LIN {X 0,Y 312.63,Z 536.352,A -85,B 0,C 180,E1 -15641.656,E2 -15641.656} C_VEL
LIN {X 0,Y 312.686,Z 536.349,A -85,B 0,C 180,E1 -15645.686,E2 -15645.686} C_VEL
LIN {X 0,Y 312.696,Z 536.347,A -85,B 0,C 180,E1 -15649.642,E2 -15649.642} C_VEL
LIN {X 0,Y 312.865,Z 536.328,A -85,B 0,C 180,E1 -15652.255,E2 -15652.255} C_VEL
LIN {X 0,Y 312.73,Z 536.383,A -85,B 0,C 180,E1 -15655.005,E2 -15655.005} C_VEL
LIN {X 0,Y 312.813,Z 536.954,A -85,B 0,C 180,E1 -15655.329,E2 -15655.329} C_VEL
LIN {X 0,Y 313.996,Z 539.629,A -85,B 0,C 180,E1 -15655.654,E2 -15655.654} C_VEL
LIN {X 0,Y 315.234,Z 541.537,A -85,B 0,C 180,E1 -15655.877,E2 -15655.877} C_VEL
LIN {X 0,Y 320.48,Z 550.525,A -85,B 0,C 180,E1 -15656.823,E2 -15656.823} C_VEL
LIN {X 0,Y 324.46,Z 558.584,A -85,B 0,C 180,E1 -15657.53,E2 -15657.53} C_VEL
LIN {X 0,Y 325.877,Z 561.864,A -85,B 0,C 180,E1 -15657.785,E2 -15657.785} C_VEL
LIN {X 0,Y 325.89,Z 581.398,A -85,B 0,C 180,E1 -15658.425,E2 -15658.425} C_VEL
LIN {X 0,Y 325.629,Z 593.005,A -85,B 0,C 180,E1 -15659.034,E2 -15659.034} C_VEL
LIN {X 0,Y 325.007,Z 604.189,A -85,B 0,C 180,E1 -15659.846,E2 -15659.846} C_VEL
LIN {X 0,Y 323.968,Z 615.161,A -85,B 0,C 180,E1 -15660.872,E2 -15660.872} C_VEL
LIN {X 0,Y 322.791,Z 625.783,A -85,B 0,C 180,E1 -15662.153,E2 -15662.153} C_VEL
LIN {X 0,Y 321.588,Z 634.422,A -85,B 0,C 180,E1 -15663.446,E2 -15663.446} C_VEL
LIN {X 0,Y 320.193,Z 643.041,A -85,B 0,C 180,E1 -15665.037,E2 -15665.037} C_VEL
LIN {X 0,Y 318.928,Z 650.052,A -85,B 0,C 180,E1 -15666.64,E2 -15666.64} C_VEL
LIN {X 0,Y 317.7,Z 655.851,A -85,B 0,C 180,E1 -15668.268,E2 -15668.268} C_VEL
LIN {X 0,Y 316.44,Z 661.361,A -85,B 0,C 180,E1 -15670.235,E2 -15670.235} C_VEL
LIN {X 0,Y 315.396,Z 665.429,A -85,B 0,C 180,E1 -15672.157,E2 -15672.157} C_VEL
LIN {X 0,Y 314.468,Z 668.571,A -85,B 0,C 180,E1 -15674.232,E2 -15674.232} C_VEL
LIN {X 0,Y 313.936,Z 670.088,A -85,B 0,C 180,E1 -15675.719,E2 -15675.719} C_VEL
LIN {X 0,Y 313.56,Z 670.868,A -85,B 0,C 180,E1 -15676.941,E2 -15676.941} C_VEL
LIN {X 0,Y 313.238,Z 671.303,A -85,B 0,C 180,E1 -15678.308,E2 -15678.308} C_VEL
LIN {X 0,Y 313.012,Z 671.234,A -85,B 0,C 180,E1 -15679.682,E2 -15679.682} C_VEL
LIN {X 0,Y 312.851,Z 670.681,A -85,B 0,C 180,E1 -15681.066,E2 -15681.066} C_VEL
LIN {X 0,Y 312.748,Z 669.215,A -85,B 0,C 180,E1 -15682.881,E2 -15682.881} C_VEL
LIN {X 0,Y 312.895,Z 665.987,A -85,B 0,C 180,E1 -15685.263,E2 -15685.263} C_VEL
LIN {X 0,Y 313.204,Z 661.722,A -85,B 0,C 180,E1 -15687.388,E2 -15687.388} C_VEL
LIN {X 0,Y 313.668,Z 655.995,A -85,B 0,C 180,E1 -15689.534,E2 -15689.534} C_VEL
LIN {X 0,Y 314.243,Z 649.623,A -85,B 0,C 180,E1 -15691.402,E2 -15691.402} C_VEL
LIN {X 0,Y 314.858,Z 642.22,A -85,B 0,C 180,E1 -15693.153,E2 -15693.153} C_VEL
LIN {X 0,Y 315.63,Z 633.354,A -85,B 0,C 180,E1 -15694.86,E2 -15694.86} C_VEL
LIN {X 0,Y 316.364,Z 624.447,A -85,B 0,C 180,E1 -15696.262,E2 -15696.262} C_VEL
LIN {X 0,Y 317.032,Z 614.062,A -85,B 0,C 180,E1 -15697.592,E2 -15697.592} C_VEL
LIN {X 0,Y 317.81,Z 601.895,A -85,B 0,C 180,E1 -15698.818,E2 -15698.818} C_VEL
LIN {X 0,Y 318.333,Z 589.989,A -85,B 0,C 180,E1 -15699.733,E2 -15699.733} C_VEL
LIN {X 0,Y 318.574,Z 576.988,A -85,B 0,C 180,E1 -15700.458,E2 -15700.458} C_VEL
LIN {X 0,Y 318.669,Z 563.154,A -85,B 0,C 180,E1 -15700.946,E2 -15700.946} C_VEL
LIN {X 0,Y 318.586,Z 555.236,A -85,B 0,C 180,E1 -15701.168,E2 -15701.168} C_VEL
LIN {X 0,Y 312.709,Z 537.424,A -85,B 0,C 180,E1 -15701.948,E2 -15701.948} C_VEL
LIN {X 0,Y 312.51,Z 536.496,A -85,B 0,C 180,E1 -15702.177,E2 -15702.177} C_VEL
LIN {X 0,Y 312.536,Z 536.364,A -85,B 0,C 180,E1 -15706.021,E2 -15706.021} C_VEL
LIN {X 0,Y 312.53,Z 536.366,A -85,B 0,C 180,E1 -15709.87,E2 -15709.87} C_VEL
LIN {X 0,Y 312.552,Z 536.362,A -85,B 0,C 180,E1 -15712.62,E2 -15712.62} C_VEL
LIN {X 0,Y 312.52,Z 536.366,A -85,B 0,C 180,E1 -15716.312,E2 -15716.312} C_VEL
LIN {X 0,Y 312.547,Z 536.362,A -85,B 0,C 180,E1 -15720.351,E2 -15720.351} C_VEL
LIN {X 0,Y 312.605,Z 536.356,A -85,B 0,C 180,E1 -15724.065,E2 -15724.065} C_VEL
LIN {X 0,Y 312.59,Z 536.362,A -85,B 0,C 180,E1 -15727.53,E2 -15727.53} C_VEL
LIN {X 0,Y 312.585,Z 536.362,A -85,B 0,C 180,E1 -15731.654,E2 -15731.654} C_VEL
LIN {X 0,Y 312.689,Z 536.349,A -85,B 0,C 180,E1 -15735.686,E2 -15735.686} C_VEL
LIN {X 0,Y 312.702,Z 536.349,A -85,B 0,C 180,E1 -15739.642,E2 -15739.642} C_VEL
LIN {X 0,Y 312.821,Z 536.328,A -85,B 0,C 180,E1 -15742.253,E2 -15742.253} C_VEL
LIN {X 0,Y 312.71,Z 536.342,A -85,B 0,C 180,E1 -15744.842,E2 -15744.842} C_VEL
LIN {X 0,Y 312.993,Z 536.306,A -85,B 0,C 180,E1 -15748.713,E2 -15748.713} C_VEL
LIN {X 0,Y 312.993,Z 536.308,A -85,B 0,C 180,E1 -15751.287,E2 -15751.287} C_VEL
LIN {X 0,Y 312.71,Z 536.342,A -85,B 0,C 180,E1 -15755.158,E2 -15755.158} C_VEL
LIN {X 0,Y 312.822,Z 536.333,A -85,B 0,C 180,E1 -15757.747,E2 -15757.747} C_VEL
LIN {X 0,Y 312.668,Z 536.351,A -85,B 0,C 180,E1 -15761.671,E2 -15761.671} C_VEL
LIN {X 0,Y 312.704,Z 536.342,A -85,B 0,C 180,E1 -15764.887,E2 -15764.887} C_VEL
LIN {X 0,Y 312.633,Z 536.352,A -85,B 0,C 180,E1 -15769.235,E2 -15769.235} C_VEL
LIN {X 0,Y 312.529,Z 536.364,A -85,B 0,C 180,E1 -15772.78,E2 -15772.78} C_VEL
LIN {X 0,Y 312.605,Z 536.361,A -85,B 0,C 180,E1 -15775.935,E2 -15775.935} C_VEL
LIN {X 0,Y 312.54,Z 536.365,A -85,B 0,C 180,E1 -15779.65,E2 -15779.65} C_VEL
LIN {X 0,Y 312.521,Z 536.368,A -85,B 0,C 180,E1 -15783.688,E2 -15783.688} C_VEL
LIN {X 0,Y 312.553,Z 536.361,A -85,B 0,C 180,E1 -15787.38,E2 -15787.38} C_VEL
LIN {X 0,Y 312.533,Z 536.365,A -85,B 0,C 180,E1 -15790.701,E2 -15790.701} C_VEL
LIN {X 0,Y 312.536,Z 536.368,A -85,B 0,C 180,E1 -15794.193,E2 -15794.193} C_VEL
LIN {X 0,Y 312.485,Z 536.373,A -85,B 0,C 180,E1 -15797.917,E2 -15797.917} C_VEL
LIN {X 0,Y 312.532,Z 536.367,A -85,B 0,C 180,E1 -15801.909,E2 -15801.909} C_VEL
LIN {X 0,Y 312.504,Z 536.369,A -85,B 0,C 180,E1 -15805.789,E2 -15805.789} C_VEL
LIN {X 0,Y 312.525,Z 536.365,A -85,B 0,C 180,E1 -15808.853,E2 -15808.853} C_VEL
LIN {X 0,Y 312.543,Z 536.361,A -85,B 0,C 180,E1 -15812.28,E2 -15812.28} C_VEL
LIN {X 0,Y 312.581,Z 536.359,A -85,B 0,C 180,E1 -15814.71,E2 -15814.71} C_VEL
LIN {X 0,Y 312.559,Z 536.359,A -85,B 0,C 180,E1 -15817.877,E2 -15817.877} C_VEL
LIN {X 0,Y 311.858,Z 536.449,A -85,B 0,C 180,E1 -15818.953,E2 -15818.953} C_VEL
LIN {X 0,Y 309.002,Z 536.806,A -85,B 0,C 180,E1 -15820.705,E2 -15820.705} C_VEL
LIN {X 0,Y 306.622,Z 537.103,A -85,B 0,C 180,E1 -15822.125,E2 -15822.125} C_VEL
LIN {X 0,Y 305.631,Z 537.223,A -85,B 0,C 180,E1 -15823.225,E2 -15823.225} C_VEL
LIN {X 0,Y 305.566,Z 537.232,A -85,B 0,C 180,E1 -15823.597,E2 -15823.597} C_VEL
LIN {X 0,Y 305.585,Z 537.232,A -85,B 0,C 180,E1 -15826.703,E2 -15826.703} C_VEL
LIN {X 0,Y 305.791,Z 537.203,A -85,B 0,C 180,E1 -15831.207,E2 -15831.207} C_VEL
LIN {X 0,Y 305.847,Z 537.196,A -85,B 0,C 180,E1 -15833.402,E2 -15833.402} C_VEL
LIN {X 0,Y 305.951,Z 537.187,A -85,B 0,C 180,E1 -15838.683,E2 -15838.683} C_VEL
LIN {X 0,Y 305.95,Z 537.184,A -85,B 0,C 180,E1 -15841.316,E2 -15841.316} C_VEL
LIN {X 0,Y 305.682,Z 537.218,A -85,B 0,C 180,E1 -15845.276,E2 -15845.276} C_VEL
LIN {X 0,Y 305.802,Z 537.203,A -85,B 0,C 180,E1 -15847.926,E2 -15847.926} C_VEL
LIN {X 0,Y 305.596,Z 537.228,A -85,B 0,C 180,E1 -15851.945,E2 -15851.945} C_VEL
LIN {X 0,Y 305.631,Z 537.225,A -85,B 0,C 180,E1 -15855.034,E2 -15855.034} C_VEL
LIN {X 0,Y 305.573,Z 537.235,A -85,B 0,C 180,E1 -15858.783,E2 -15858.783} C_VEL
LIN {X 0,Y 305.48,Z 537.245,A -85,B 0,C 180,E1 -15863.039,E2 -15863.039} C_VEL
LIN {X 0,Y 305.548,Z 537.235,A -85,B 0,C 180,E1 -15866.229,E2 -15866.229} C_VEL
LIN {X 0,Y 305.49,Z 537.244,A -85,B 0,C 180,E1 -15869.05,E2 -15869.05} C_VEL
LIN {X 0,Y 305.459,Z 537.245,A -85,B 0,C 180,E1 -15873.517,E2 -15873.517} C_VEL
LIN {X 0,Y 305.467,Z 537.249,A -85,B 0,C 180,E1 -15876.74,E2 -15876.74} C_VEL
LIN {X 0,Y 305.449,Z 537.25,A -85,B 0,C 180,E1 -15880.6,E2 -15880.6} C_VEL
LIN {X 0,Y 305.414,Z 537.253,A -85,B 0,C 180,E1 -15884.493,E2 -15884.493} C_VEL
LIN {X 0,Y 305.438,Z 537.248,A -85,B 0,C 180,E1 -15888.144,E2 -15888.144} C_VEL
LIN {X 0,Y 305.472,Z 537.244,A -85,B 0,C 180,E1 -15891.598,E2 -15891.598} C_VEL
LIN {X 0,Y 305.61,Z 537.416,A -85,B 0,C 180,E1 -15894.301,E2 -15894.301} C_VEL
LIN {X 0,Y 308.315,Z 551.362,A -85,B 0,C 180,E1 -15898.752,E2 -15898.752} C_VEL
LIN {X 0,Y 309.128,Z 556.658,A -85,B 0,C 180,E1 -15900.365,E2 -15900.365} C_VEL
LIN {X 0,Y 307.296,Z 571.295,A -85,B 0,C 180,E1 -15904.608,E2 -15904.608} C_VEL
LIN {X 0,Y 305.685,Z 588.18,A -85,B 0,C 180,E1 -15909.476,E2 -15909.476} C_VEL
LIN {X 0,Y 305.517,Z 589.903,A -85,B 0,C 180,E1 -15909.891,E2 -15909.891} C_VEL
LIN {X 0,Y 309.829,Z 651.427,A -85,B 0,C 180,E1 -15912.133,E2 -15912.133} C_VEL
LIN {X 0,Y 309.126,Z 676.197,A -85,B 0,C 180,E1 -15912.98,E2 -15912.98} C_VEL
LIN {X 0,Y 308.596,Z 687.867,A -85,B 0,C 180,E1 -15913.631,E2 -15913.631} C_VEL
LIN {X 0,Y 307.713,Z 698.277,A -85,B 0,C 180,E1 -15914.433,E2 -15914.433} C_VEL
LIN {X 0,Y 306.771,Z 709.39,A -85,B 0,C 180,E1 -15915.574,E2 -15915.574} C_VEL
LIN {X 0,Y 306.007,Z 719.359,A -85,B 0,C 180,E1 -15916.892,E2 -15916.892} C_VEL
LIN {X 0,Y 305.232,Z 728.218,A -85,B 0,C 180,E1 -15918.377,E2 -15918.377} C_VEL
LIN {X 0,Y 304.777,Z 736.134,A -85,B 0,C 180,E1 -15920.041,E2 -15920.041} C_VEL
LIN {X 0,Y 304.572,Z 742.449,A -85,B 0,C 180,E1 -15921.708,E2 -15921.708} C_VEL
LIN {X 0,Y 304.624,Z 747.486,A -85,B 0,C 180,E1 -15923.376,E2 -15923.376} C_VEL
LIN {X 0,Y 304.895,Z 752.023,A -85,B 0,C 180,E1 -15925.373,E2 -15925.373} C_VEL
LIN {X 0,Y 305.09,Z 755.096,A -85,B 0,C 180,E1 -15927.359,E2 -15927.359} C_VEL
LIN {X 0,Y 305.334,Z 756.407,A -85,B 0,C 180,E1 -15928.681,E2 -15928.681} C_VEL
LIN {X 0,Y 305.562,Z 757.164,A -85,B 0,C 180,E1 -15930,E2 -15930} C_VEL
LIN {X 0,Y 305.109,Z 757.234,A -85,B 0,C 180,E1 -15931.32,E2 -15931.32} C_VEL
LIN {X 0,Y 304.892,Z 756.821,A -85,B 0,C 180,E1 -15932.642,E2 -15932.642} C_VEL
LIN {X 0,Y 304.681,Z 755.839,A -85,B 0,C 180,E1 -15933.968,E2 -15933.968} C_VEL
LIN {X 0,Y 304.419,Z 754.339,A -85,B 0,C 180,E1 -15935.298,E2 -15935.298} C_VEL
LIN {X 0,Y 304.248,Z 751.04,A -85,B 0,C 180,E1 -15937.299,E2 -15937.299} C_VEL
LIN {X 0,Y 304.4,Z 746.467,A -85,B 0,C 180,E1 -15939.3,E2 -15939.3} C_VEL
LIN {X 0,Y 304.897,Z 740.46,A -85,B 0,C 180,E1 -15941.299,E2 -15941.299} C_VEL
LIN {X 0,Y 305.993,Z 732.774,A -85,B 0,C 180,E1 -15943.278,E2 -15943.278} C_VEL
LIN {X 0,Y 307.358,Z 724.75,A -85,B 0,C 180,E1 -15944.906,E2 -15944.906} C_VEL
LIN {X 0,Y 308.946,Z 714.928,A -85,B 0,C 180,E1 -15946.52,E2 -15946.52} C_VEL
LIN {X 0,Y 310.94,Z 703.756,A -85,B 0,C 180,E1 -15947.936,E2 -15947.936} C_VEL
LIN {X 0,Y 312.695,Z 691.885,A -85,B 0,C 180,E1 -15949.096,E2 -15949.096} C_VEL
LIN {X 0,Y 314.143,Z 680.329,A -85,B 0,C 180,E1 -15949.948,E2 -15949.948} C_VEL
LIN {X 0,Y 315.4,Z 667.35,A -85,B 0,C 180,E1 -15950.63,E2 -15950.63} C_VEL
LIN {X 0,Y 316.09,Z 651.138,A -85,B 0,C 180,E1 -15951.19,E2 -15951.19} C_VEL
LIN {X 0,Y 315.177,Z 625.529,A -85,B 0,C 180,E1 -15952.203,E2 -15952.203} C_VEL
LIN {X 0,Y 313.343,Z 607.824,A -85,B 0,C 180,E1 -15953.06,E2 -15953.06} C_VEL
LIN {X 0,Y 310.491,Z 589.45,A -85,B 0,C 180,E1 -15954.097,E2 -15954.097} C_VEL
LIN {X 0,Y 307.119,Z 572.651,A -85,B 0,C 180,E1 -15955.24,E2 -15955.24} C_VEL
LIN {X 0,Y 307.26,Z 570.491,A -85,B 0,C 180,E1 -15955.758,E2 -15955.758} C_VEL
LIN {X 0,Y 309.042,Z 557.571,A -85,B 0,C 180,E1 -15959.644,E2 -15959.644} C_VEL
LIN {X 0,Y 309.131,Z 555.676,A -85,B 0,C 180,E1 -15960.241,E2 -15960.241} C_VEL
LIN {X 0,Y 307.588,Z 547.039,A -85,B 0,C 180,E1 -15963.254,E2 -15963.254} C_VEL
LIN {X 0,Y 305.816,Z 538.651,A -85,B 0,C 180,E1 -15966.454,E2 -15966.454} C_VEL
LIN {X 0,Y 305.495,Z 537.259,A -85,B 0,C 180,E1 -15967.148,E2 -15967.148} C_VEL
LIN {X 0,Y 305.45,Z 537.248,A -85,B 0,C 180,E1 -15970.599,E2 -15970.599} C_VEL
LIN {X 0,Y 305.456,Z 537.244,A -85,B 0,C 180,E1 -15974.5,E2 -15974.5} C_VEL
LIN {X 0,Y 305.49,Z 537.236,A -85,B 0,C 180,E1 -15978.152,E2 -15978.152} C_VEL
LIN {X 0,Y 305.516,Z 537.236,A -85,B 0,C 180,E1 -15981.604,E2 -15981.604} C_VEL
LIN {X 0,Y 305.457,Z 537.243,A -85,B 0,C 180,E1 -15984.887,E2 -15984.887} C_VEL
LIN {X 0,Y 305.45,Z 537.246,A -85,B 0,C 180,E1 -15988.353,E2 -15988.353} C_VEL
LIN {X 0,Y 305.514,Z 537.236,A -85,B 0,C 180,E1 -15991.114,E2 -15991.114} C_VEL
LIN {X 0,Y 305.564,Z 537.228,A -85,B 0,C 180,E1 -15994.088,E2 -15994.088} C_VEL
LIN {X 0,Y 305.518,Z 537.243,A -85,B 0,C 180,E1 -15998.405,E2 -15998.405} C_VEL
LIN {X 0,Y 305.582,Z 537.233,A -85,B 0,C 180,E1 -16001.218,E2 -16001.218} C_VEL
LIN {X 0,Y 305.642,Z 537.224,A -85,B 0,C 180,E1 -16005.349,E2 -16005.349} C_VEL
LIN {X 0,Y 305.633,Z 537.226,A -85,B 0,C 180,E1 -16009.4,E2 -16009.4} C_VEL
LIN {X 0,Y 305.806,Z 537.209,A -85,B 0,C 180,E1 -16012.075,E2 -16012.075} C_VEL
LIN {X 0,Y 305.788,Z 537.423,A -85,B 0,C 180,E1 -16014.23,E2 -16014.23} C_VEL
LIN {X 0,Y 306.003,Z 538.467,A -85,B 0,C 180,E1 -16014.482,E2 -16014.482} C_VEL
LIN {X 0,Y 307.548,Z 541.21,A -85,B 0,C 180,E1 -16014.816,E2 -16014.816} C_VEL
LIN {X 0,Y 315.14,Z 554.13,A -85,B 0,C 180,E1 -16016.28,E2 -16016.28} C_VEL
LIN {X 0,Y 319.195,Z 562.569,A -85,B 0,C 180,E1 -16017.048,E2 -16017.048} C_VEL
LIN {X 0,Y 319.98,Z 564.66,A -85,B 0,C 180,E1 -16017.207,E2 -16017.207} C_VEL
LIN {X 0,Y 319.783,Z 583.237,A -85,B 0,C 180,E1 -16017.83,E2 -16017.83} C_VEL
LIN {X 0,Y 319.495,Z 595.045,A -85,B 0,C 180,E1 -16018.48,E2 -16018.48} C_VEL
LIN {X 0,Y 318.734,Z 606.808,A -85,B 0,C 180,E1 -16019.369,E2 -16019.369} C_VEL
LIN {X 0,Y 317.66,Z 617.762,A -85,B 0,C 180,E1 -16020.445,E2 -16020.445} C_VEL
LIN {X 0,Y 316.271,Z 628.744,A -85,B 0,C 180,E1 -16021.847,E2 -16021.847} C_VEL
LIN {X 0,Y 314.988,Z 637.224,A -85,B 0,C 180,E1 -16023.198,E2 -16023.198} C_VEL
LIN {X 0,Y 313.504,Z 645.53,A -85,B 0,C 180,E1 -16024.823,E2 -16024.823} C_VEL
LIN {X 0,Y 311.884,Z 653.43,A -85,B 0,C 180,E1 -16026.772,E2 -16026.772} C_VEL
LIN {X 0,Y 310.642,Z 658.865,A -85,B 0,C 180,E1 -16028.457,E2 -16028.457} C_VEL
LIN {X 0,Y 309.372,Z 663.964,A -85,B 0,C 180,E1 -16030.471,E2 -16030.471} C_VEL
LIN {X 0,Y 308.274,Z 667.778,A -85,B 0,C 180,E1 -16032.509,E2 -16032.509} C_VEL
LIN {X 0,Y 307.341,Z 670.417,A -85,B 0,C 180,E1 -16034.569,E2 -16034.569} C_VEL
LIN {X 0,Y 306.863,Z 671.556,A -85,B 0,C 180,E1 -16035.953,E2 -16035.953} C_VEL
LIN {X 0,Y 306.466,Z 672.239,A -85,B 0,C 180,E1 -16037.345,E2 -16037.345} C_VEL
LIN {X 0,Y 305.989,Z 672.269,A -85,B 0,C 180,E1 -16039.666,E2 -16039.666} C_VEL
LIN {X 0,Y 305.78,Z 671.318,A -85,B 0,C 180,E1 -16041.577,E2 -16041.577} C_VEL
LIN {X 0,Y 305.721,Z 669.883,A -85,B 0,C 180,E1 -16043.146,E2 -16043.146} C_VEL
LIN {X 0,Y 305.846,Z 667.094,A -85,B 0,C 180,E1 -16045.158,E2 -16045.158} C_VEL
LIN {X 0,Y 306.167,Z 662.831,A -85,B 0,C 180,E1 -16047.329,E2 -16047.329} C_VEL
LIN {X 0,Y 306.592,Z 657.404,A -85,B 0,C 180,E1 -16049.419,E2 -16049.419} C_VEL
LIN {X 0,Y 307.165,Z 650.979,A -85,B 0,C 180,E1 -16051.368,E2 -16051.368} C_VEL
LIN {X 0,Y 307.817,Z 643.311,A -85,B 0,C 180,E1 -16053.228,E2 -16053.228} C_VEL
LIN {X 0,Y 308.674,Z 633.551,A -85,B 0,C 180,E1 -16055.133,E2 -16055.133} C_VEL
LIN {X 0,Y 309.592,Z 622.854,A -85,B 0,C 180,E1 -16056.78,E2 -16056.78} C_VEL
LIN {X 0,Y 310.269,Z 612.085,A -85,B 0,C 180,E1 -16058.116,E2 -16058.116} C_VEL
LIN {X 0,Y 310.974,Z 600.262,A -85,B 0,C 180,E1 -16059.258,E2 -16059.258} C_VEL
LIN {X 0,Y 311.422,Z 588.721,A -85,B 0,C 180,E1 -16060.114,E2 -16060.114} C_VEL
LIN {X 0,Y 311.681,Z 575.777,A -85,B 0,C 180,E1 -16060.806,E2 -16060.806} C_VEL
LIN {X 0,Y 311.662,Z 556.495,A -85,B 0,C 180,E1 -16061.429,E2 -16061.429} C_VEL
LIN {X 0,Y 305.662,Z 538.299,A -85,B 0,C 180,E1 -16062.251,E2 -16062.251} C_VEL
LIN {X 0,Y 305.469,Z 537.331,A -85,B 0,C 180,E1 -16062.517,E2 -16062.517} C_VEL
LIN {X 0,Y 305.492,Z 537.242,A -85,B 0,C 180,E1 -16066.358,E2 -16066.358} C_VEL
LIN {X 0,Y 305.484,Z 537.244,A -85,B 0,C 180,E1 -16069.898,E2 -16069.898} C_VEL
LIN {X 0,Y 305.502,Z 537.244,A -85,B 0,C 180,E1 -16073.627,E2 -16073.627} C_VEL
LIN {X 0,Y 305.465,Z 537.244,A -85,B 0,C 180,E1 -16076.484,E2 -16076.484} C_VEL
LIN {X 0,Y 305.497,Z 537.241,A -85,B 0,C 180,E1 -16080.951,E2 -16080.951} C_VEL
LIN {X 0,Y 305.574,Z 537.232,A -85,B 0,C 180,E1 -16084.089,E2 -16084.089} C_VEL
LIN {X 0,Y 305.497,Z 537.24,A -85,B 0,C 180,E1 -16088.403,E2 -16088.403} C_VEL
LIN {X 0,Y 305.546,Z 537.236,A -85,B 0,C 180,E1 -16091.215,E2 -16091.215} C_VEL
LIN {X 0,Y 305.63,Z 537.226,A -85,B 0,C 180,E1 -16095.349,E2 -16095.349} C_VEL
LIN {X 0,Y 305.639,Z 537.226,A -85,B 0,C 180,E1 -16099.4,E2 -16099.4} C_VEL
LIN {X 0,Y 305.768,Z 537.208,A -85,B 0,C 180,E1 -16102.073,E2 -16102.073} C_VEL
LIN {X 0,Y 305.678,Z 537.217,A -85,B 0,C 180,E1 -16104.724,E2 -16104.724} C_VEL
LIN {X 0,Y 305.96,Z 537.182,A -85,B 0,C 180,E1 -16108.684,E2 -16108.684} C_VEL
LIN {X 0,Y 305.96,Z 537.184,A -85,B 0,C 180,E1 -16111.316,E2 -16111.316} C_VEL
LIN {X 0,Y 305.679,Z 537.219,A -85,B 0,C 180,E1 -16115.277,E2 -16115.277} C_VEL
LIN {X 0,Y 305.768,Z 537.211,A -85,B 0,C 180,E1 -16117.927,E2 -16117.927} C_VEL
LIN {X 0,Y 305.603,Z 537.232,A -85,B 0,C 180,E1 -16121.945,E2 -16121.945} C_VEL
LIN {X 0,Y 305.642,Z 537.222,A -85,B 0,C 180,E1 -16125.035,E2 -16125.035} C_VEL
LIN {X 0,Y 305.579,Z 537.231,A -85,B 0,C 180,E1 -16129.444,E2 -16129.444} C_VEL
LIN {X 0,Y 305.489,Z 537.241,A -85,B 0,C 180,E1 -16133.039,E2 -16133.039} C_VEL
LIN {X 0,Y 305.534,Z 537.238,A -85,B 0,C 180,E1 -16136.22,E2 -16136.22} C_VEL
LIN {X 0,Y 305.49,Z 537.241,A -85,B 0,C 180,E1 -16139.046,E2 -16139.046} C_VEL
LIN {X 0,Y 305.445,Z 537.252,A -85,B 0,C 180,E1 -16141.951,E2 -16141.951} C_VEL
LIN {X 0,Y 305.463,Z 537.244,A -85,B 0,C 180,E1 -16145.112,E2 -16145.112} C_VEL
LIN {X 0,Y 305.494,Z 537.242,A -85,B 0,C 180,E1 -16148.538,E2 -16148.538} C_VEL
LIN {X 0,Y 305.51,Z 537.24,A -85,B 0,C 180,E1 -16152.596,E2 -16152.596} C_VEL
LIN {X 0,Y 305.466,Z 537.247,A -85,B 0,C 180,E1 -16156.351,E2 -16156.351} C_VEL
LIN {X 0,Y 305.456,Z 537.248,A -85,B 0,C 180,E1 -16159.891,E2 -16159.891} C_VEL
LIN {X 0,Y 305.481,Z 537.243,A -85,B 0,C 180,E1 -16163.63,E2 -16163.63} C_VEL
LIN {X 0,Y 305.463,Z 537.247,A -85,B 0,C 180,E1 -16166.482,E2 -16166.482} C_VEL
LIN {X 0,Y 305.463,Z 537.245,A -85,B 0,C 180,E1 -16169.59,E2 -16169.59} C_VEL
LIN {X 0,Y 305.518,Z 537.24,A -85,B 0,C 180,E1 -16172.608,E2 -16172.608} C_VEL
LIN {X 0,Y 305.504,Z 537.239,A -85,B 0,C 180,E1 -16175.538,E2 -16175.538} C_VEL
LIN {X 0,Y 305.525,Z 537.238,A -85,B 0,C 180,E1 -16179.815,E2 -16179.815} C_VEL
LIN {X 0,Y 305.57,Z 537.234,A -85,B 0,C 180,E1 -16182.602,E2 -16182.602} C_VEL
LIN {X 0,Y 305.566,Z 537.232,A -85,B 0,C 180,E1 -16183.597,E2 -16183.597} C_VEL
LIN {X 0,Y 304.937,Z 537.314,A -85,B 0,C 180,E1 -16184.697,E2 -16184.697} C_VEL
LIN {X 0,Y 302.1,Z 537.668,A -85,B 0,C 180,E1 -16186.488,E2 -16186.488} C_VEL
LIN {X 0,Y 299.685,Z 537.967,A -85,B 0,C 180,E1 -16187.94,E2 -16187.94} C_VEL
LIN {X 0,Y 298.666,Z 538.092,A -85,B 0,C 180,E1 -16189.066,E2 -16189.066} C_VEL
LIN {X 0,Y 298.594,Z 538.099,A -85,B 0,C 180,E1 -16189.447,E2 -16189.447} C_VEL
LIN {X 0,Y 298.753,Z 538.081,A -85,B 0,C 180,E1 -16191.885,E2 -16191.885} C_VEL
LIN {X 0,Y 298.655,Z 538.097,A -85,B 0,C 180,E1 -16194.598,E2 -16194.598} C_VEL
LIN {X 0,Y 298.917,Z 538.063,A -85,B 0,C 180,E1 -16198.652,E2 -16198.652} C_VEL
LIN {X 0,Y 298.917,Z 538.06,A -85,B 0,C 180,E1 -16201.347,E2 -16201.347} C_VEL
LIN {X 0,Y 298.786,Z 538.079,A -85,B 0,C 180,E1 -16206.754,E2 -16206.754} C_VEL
LIN {X 0,Y 298.674,Z 538.089,A -85,B 0,C 180,E1 -16209.48,E2 -16209.48} C_VEL
LIN {X 0,Y 298.545,Z 538.106,A -85,B 0,C 180,E1 -16213.615,E2 -16213.615} C_VEL
LIN {X 0,Y 298.542,Z 538.11,A -85,B 0,C 180,E1 -16216.409,E2 -16216.409} C_VEL
LIN {X 0,Y 298.492,Z 538.112,A -85,B 0,C 180,E1 -16219.647,E2 -16219.647} C_VEL
LIN {X 0,Y 298.423,Z 538.122,A -85,B 0,C 180,E1 -16223.6,E2 -16223.6} C_VEL
LIN {X 0,Y 298.486,Z 538.117,A -85,B 0,C 180,E1 -16226.574,E2 -16226.574} C_VEL
LIN {X 0,Y 298.415,Z 538.122,A -85,B 0,C 180,E1 -16229.641,E2 -16229.641} C_VEL
LIN {X 0,Y 298.39,Z 538.131,A -85,B 0,C 180,E1 -16232.8,E2 -16232.8} C_VEL
LIN {X 0,Y 298.439,Z 538.124,A -85,B 0,C 180,E1 -16236.807,E2 -16236.807} C_VEL
LIN {X 0,Y 298.383,Z 538.13,A -85,B 0,C 180,E1 -16241.088,E2 -16241.088} C_VEL
LIN {X 0,Y 298.384,Z 538.13,A -85,B 0,C 180,E1 -16245.042,E2 -16245.042} C_VEL
LIN {X 0,Y 298.384,Z 538.132,A -85,B 0,C 180,E1 -16248.912,E2 -16248.912} C_VEL
LIN {X 0,Y 298.475,Z 538.12,A -85,B 0,C 180,E1 -16253.185,E2 -16253.185} C_VEL
LIN {X 0,Y 298.562,Z 538.263,A -85,B 0,C 180,E1 -16254.129,E2 -16254.129} C_VEL
LIN {X 0,Y 301.267,Z 552.322,A -85,B 0,C 180,E1 -16258.732,E2 -16258.732} C_VEL
LIN {X 0,Y 302.049,Z 556.84,A -85,B 0,C 180,E1 -16260.148,E2 -16260.148} C_VEL
LIN {X 0,Y 300.448,Z 569.706,A -85,B 0,C 180,E1 -16263.986,E2 -16263.986} C_VEL
LIN {X 0,Y 298.8,Z 585.325,A -85,B 0,C 180,E1 -16268.619,E2 -16268.619} C_VEL
LIN {X 0,Y 298.551,Z 588.735,A -85,B 0,C 180,E1 -16269.546,E2 -16269.546} C_VEL
LIN {X 0,Y 302.841,Z 651.586,A -85,B 0,C 180,E1 -16271.899,E2 -16271.899} C_VEL
LIN {X 0,Y 302.123,Z 675.368,A -85,B 0,C 180,E1 -16272.747,E2 -16272.747} C_VEL
LIN {X 0,Y 301.618,Z 686.939,A -85,B 0,C 180,E1 -16273.415,E2 -16273.415} C_VEL
LIN {X 0,Y 300.747,Z 697.315,A -85,B 0,C 180,E1 -16274.237,E2 -16274.237} C_VEL
LIN {X 0,Y 299.754,Z 708.387,A -85,B 0,C 180,E1 -16275.402,E2 -16275.402} C_VEL
LIN {X 0,Y 299.076,Z 717.224,A -85,B 0,C 180,E1 -16276.582,E2 -16276.582} C_VEL
LIN {X 0,Y 298.264,Z 726.3,A -85,B 0,C 180,E1 -16278.102,E2 -16278.102} C_VEL
LIN {X 0,Y 297.75,Z 734.414,A -85,B 0,C 180,E1 -16279.803,E2 -16279.803} C_VEL
LIN {X 0,Y 297.534,Z 742,A -85,B 0,C 180,E1 -16281.852,E2 -16281.852} C_VEL
LIN {X 0,Y 297.663,Z 747.732,A -85,B 0,C 180,E1 -16283.901,E2 -16283.901} C_VEL
LIN {X 0,Y 297.927,Z 751.908,A -85,B 0,C 180,E1 -16285.942,E2 -16285.942} C_VEL
LIN {X 0,Y 298.059,Z 753.847,A -85,B 0,C 180,E1 -16287.297,E2 -16287.297} C_VEL
LIN {X 0,Y 298.314,Z 755.241,A -85,B 0,C 180,E1 -16288.65,E2 -16288.65} C_VEL
LIN {X 0,Y 298.54,Z 756.035,A -85,B 0,C 180,E1 -16290,E2 -16290} C_VEL
LIN {X 0,Y 298.072,Z 756.178,A -85,B 0,C 180,E1 -16291.351,E2 -16291.351} C_VEL
LIN {X 0,Y 297.835,Z 755.797,A -85,B 0,C 180,E1 -16292.705,E2 -16292.705} C_VEL
LIN {X 0,Y 297.602,Z 754.888,A -85,B 0,C 180,E1 -16294.062,E2 -16294.062} C_VEL
LIN {X 0,Y 297.33,Z 753.432,A -85,B 0,C 180,E1 -16295.425,E2 -16295.425} C_VEL
LIN {X 0,Y 297.165,Z 750.26,A -85,B 0,C 180,E1 -16297.474,E2 -16297.474} C_VEL
LIN {X 0,Y 297.33,Z 745.776,A -85,B 0,C 180,E1 -16299.524,E2 -16299.524} C_VEL
LIN {X 0,Y 297.885,Z 739.902,A -85,B 0,C 180,E1 -16301.568,E2 -16301.568} C_VEL
LIN {X 0,Y 299.063,Z 732.406,A -85,B 0,C 180,E1 -16303.591,E2 -16303.591} C_VEL
LIN {X 0,Y 300.502,Z 724.661,A -85,B 0,C 180,E1 -16305.254,E2 -16305.254} C_VEL
LIN {X 0,Y 302.164,Z 715.054,A -85,B 0,C 180,E1 -16306.902,E2 -16306.902} C_VEL
LIN {X 0,Y 304.23,Z 704.239,A -85,B 0,C 180,E1 -16308.345,E2 -16308.345} C_VEL
LIN {X 0,Y 305.931,Z 693.671,A -85,B 0,C 180,E1 -16309.46,E2 -16309.46} C_VEL
LIN {X 0,Y 307.691,Z 681.024,A -85,B 0,C 180,E1 -16310.473,E2 -16310.473} C_VEL
LIN {X 0,Y 309.071,Z 668.287,A -85,B 0,C 180,E1 -16311.204,E2 -16311.204} C_VEL
LIN {X 0,Y 309.914,Z 655.245,A -85,B 0,C 180,E1 -16311.708,E2 -16311.708} C_VEL
LIN {X 0,Y 309.25,Z 629.64,A -85,B 0,C 180,E1 -16312.726,E2 -16312.726} C_VEL
LIN {X 0,Y 307.774,Z 612.039,A -85,B 0,C 180,E1 -16313.565,E2 -16313.565} C_VEL
LIN {X 0,Y 304.89,Z 592.145,A -85,B 0,C 180,E1 -16314.733,E2 -16314.733} C_VEL
LIN {X 0,Y 301.258,Z 574.403,A -85,B 0,C 180,E1 -16315.977,E2 -16315.977} C_VEL
LIN {X 0,Y 300.477,Z 570.14,A -85,B 0,C 180,E1 -16316.336,E2 -16316.336} C_VEL
LIN {X 0,Y 302.158,Z 558.138,A -85,B 0,C 180,E1 -16320.004,E2 -16320.004} C_VEL
LIN {X 0,Y 301.589,Z 553.455,A -85,B 0,C 180,E1 -16321.622,E2 -16321.622} C_VEL
LIN {X 0,Y 299.704,Z 543.654,A -85,B 0,C 180,E1 -16325.304,E2 -16325.304} C_VEL
LIN {X 0,Y 298.465,Z 538.144,A -85,B 0,C 180,E1 -16327.654,E2 -16327.654} C_VEL
LIN {X 0,Y 298.382,Z 538.131,A -85,B 0,C 180,E1 -16331.261,E2 -16331.261} C_VEL
LIN {X 0,Y 298.412,Z 538.12,A -85,B 0,C 180,E1 -16335.046,E2 -16335.046} C_VEL
LIN {X 0,Y 298.449,Z 538.117,A -85,B 0,C 180,E1 -16338.75,E2 -16338.75} C_VEL
LIN {X 0,Y 298.444,Z 538.121,A -85,B 0,C 180,E1 -16342.247,E2 -16342.247} C_VEL
LIN {X 0,Y 298.403,Z 538.128,A -85,B 0,C 180,E1 -16345.581,E2 -16345.581} C_VEL
LIN {X 0,Y 298.393,Z 538.128,A -85,B 0,C 180,E1 -16348.791,E2 -16348.791} C_VEL
LIN {X 0,Y 298.457,Z 538.121,A -85,B 0,C 180,E1 -16351.904,E2 -16351.904} C_VEL
LIN {X 0,Y 298.479,Z 538.117,A -85,B 0,C 180,E1 -16354.924,E2 -16354.924} C_VEL
LIN {X 0,Y 298.451,Z 538.116,A -85,B 0,C 180,E1 -16359.316,E2 -16359.316} C_VEL
LIN {X 0,Y 298.53,Z 538.106,A -85,B 0,C 180,E1 -16362.179,E2 -16362.179} C_VEL
LIN {X 0,Y 298.586,Z 538.101,A -85,B 0,C 180,E1 -16364.995,E2 -16364.995} C_VEL
LIN {X 0,Y 298.588,Z 538.103,A -85,B 0,C 180,E1 -16369.147,E2 -16369.147} C_VEL
LIN {X 0,Y 298.775,Z 538.082,A -85,B 0,C 180,E1 -16372.567,E2 -16372.567} C_VEL
LIN {X 0,Y 298.845,Z 538.428,A -85,B 0,C 180,E1 -16373.248,E2 -16373.248} C_VEL
LIN {X 0,Y 299.031,Z 539.139,A -85,B 0,C 180,E1 -16373.424,E2 -16373.424} C_VEL
LIN {X 0,Y 300.479,Z 541.9,A -85,B 0,C 180,E1 -16373.787,E2 -16373.787} C_VEL
LIN {X 0,Y 309.768,Z 557.651,A -85,B 0,C 180,E1 -16375.707,E2 -16375.707} C_VEL
LIN {X 0,Y 313.993,Z 566.485,A -85,B 0,C 180,E1 -16376.54,E2 -16376.54} C_VEL
LIN {X 0,Y 313.839,Z 584.612,A -85,B 0,C 180,E1 -16377.178,E2 -16377.178} C_VEL
LIN {X 0,Y 313.493,Z 595.952,A -85,B 0,C 180,E1 -16377.813,E2 -16377.813} C_VEL
LIN {X 0,Y 312.68,Z 607.648,A -85,B 0,C 180,E1 -16378.713,E2 -16378.713} C_VEL
LIN {X 0,Y 311.505,Z 618.915,A -85,B 0,C 180,E1 -16379.839,E2 -16379.839} C_VEL
LIN {X 0,Y 310.128,Z 629.316,A -85,B 0,C 180,E1 -16381.177,E2 -16381.177} C_VEL
LIN {X 0,Y 308.718,Z 638.236,A -85,B 0,C 180,E1 -16382.61,E2 -16382.61} C_VEL
LIN {X 0,Y 307.137,Z 646.594,A -85,B 0,C 180,E1 -16384.265,E2 -16384.265} C_VEL
LIN {X 0,Y 305.389,Z 654.567,A -85,B 0,C 180,E1 -16386.276,E2 -16386.276} C_VEL
LIN {X 0,Y 304.055,Z 659.921,A -85,B 0,C 180,E1 -16387.972,E2 -16387.972} C_VEL
LIN {X 0,Y 302.672,Z 665.029,A -85,B 0,C 180,E1 -16390.03,E2 -16390.03} C_VEL
LIN {X 0,Y 301.507,Z 668.864,A -85,B 0,C 180,E1 -16392.11,E2 -16392.11} C_VEL
LIN {X 0,Y 300.832,Z 670.739,A -85,B 0,C 180,E1 -16393.511,E2 -16393.511} C_VEL
LIN {X 0,Y 300.225,Z 672.162,A -85,B 0,C 180,E1 -16394.922,E2 -16394.922} C_VEL
LIN {X 0,Y 299.752,Z 673.05,A -85,B 0,C 180,E1 -16396.342,E2 -16396.342} C_VEL
LIN {X 0,Y 299.363,Z 673.482,A -85,B 0,C 180,E1 -16397.77,E2 -16397.77} C_VEL
LIN {X 0,Y 298.964,Z 673.231,A -85,B 0,C 180,E1 -16399.9,E2 -16399.9} C_VEL
LIN {X 0,Y 298.738,Z 671.847,A -85,B 0,C 180,E1 -16402.112,E2 -16402.112} C_VEL
LIN {X 0,Y 298.764,Z 669.297,A -85,B 0,C 180,E1 -16404.31,E2 -16404.31} C_VEL
LIN {X 0,Y 299.014,Z 665.095,A -85,B 0,C 180,E1 -16406.731,E2 -16406.731} C_VEL
LIN {X 0,Y 299.368,Z 660.302,A -85,B 0,C 180,E1 -16408.768,E2 -16408.768} C_VEL
LIN {X 0,Y 299.976,Z 653.382,A -85,B 0,C 180,E1 -16411.027,E2 -16411.027} C_VEL
LIN {X 0,Y 300.64,Z 646.242,A -85,B 0,C 180,E1 -16412.884,E2 -16412.884} C_VEL
LIN {X 0,Y 301.504,Z 636.944,A -85,B 0,C 180,E1 -16414.827,E2 -16414.827} C_VEL
LIN {X 0,Y 302.353,Z 626.597,A -85,B 0,C 180,E1 -16416.559,E2 -16416.559} C_VEL
LIN {X 0,Y 303.129,Z 615.426,A -85,B 0,C 180,E1 -16418.04,E2 -16418.04} C_VEL
LIN {X 0,Y 303.909,Z 603.571,A -85,B 0,C 180,E1 -16419.277,E2 -16419.277} C_VEL
LIN {X 0,Y 304.473,Z 591.008,A -85,B 0,C 180,E1 -16420.265,E2 -16420.265} C_VEL
LIN {X 0,Y 304.753,Z 578,A -85,B 0,C 180,E1 -16421.005,E2 -16421.005} C_VEL
LIN {X 0,Y 304.845,Z 562.247,A -85,B 0,C 180,E1 -16421.555,E2 -16421.555} C_VEL
LIN {X 0,Y 304.662,Z 557.668,A -85,B 0,C 180,E1 -16421.699,E2 -16421.699} C_VEL
LIN {X 0,Y 298.593,Z 539.09,A -85,B 0,C 180,E1 -16422.563,E2 -16422.563} C_VEL
LIN {X 0,Y 298.423,Z 538.204,A -85,B 0,C 180,E1 -16422.829,E2 -16422.829} C_VEL
LIN {X 0,Y 298.467,Z 538.119,A -85,B 0,C 180,E1 -16426.934,E2 -16426.934} C_VEL
LIN {X 0,Y 298.436,Z 538.122,A -85,B 0,C 180,E1 -16431,E2 -16431} C_VEL
LIN {X 0,Y 298.434,Z 538.122,A -85,B 0,C 180,E1 -16433.933,E2 -16433.933} C_VEL
LIN {X 0,Y 298.396,Z 538.126,A -85,B 0,C 180,E1 -16437.984,E2 -16437.984} C_VEL
LIN {X 0,Y 298.465,Z 538.118,A -85,B 0,C 180,E1 -16441.905,E2 -16441.905} C_VEL
LIN {X 0,Y 298.488,Z 538.114,A -85,B 0,C 180,E1 -16444.925,E2 -16444.925} C_VEL
LIN {X 0,Y 298.442,Z 538.122,A -85,B 0,C 180,E1 -16449.315,E2 -16449.315} C_VEL
LIN {X 0,Y 298.508,Z 538.111,A -85,B 0,C 180,E1 -16452.178,E2 -16452.178} C_VEL
LIN {X 0,Y 298.589,Z 538.101,A -85,B 0,C 180,E1 -16454.995,E2 -16454.995} C_VEL
LIN {X 0,Y 298.595,Z 538.101,A -85,B 0,C 180,E1 -16459.147,E2 -16459.147} C_VEL
LIN {X 0,Y 298.717,Z 538.088,A -85,B 0,C 180,E1 -16461.885,E2 -16461.885} C_VEL
LIN {X 0,Y 298.647,Z 538.093,A -85,B 0,C 180,E1 -16464.599,E2 -16464.599} C_VEL
LIN {X 0,Y 298.926,Z 538.059,A -85,B 0,C 180,E1 -16468.653,E2 -16468.653} C_VEL
LIN {X 0,Y 298.927,Z 538.06,A -85,B 0,C 180,E1 -16471.347,E2 -16471.347} C_VEL
LIN {X 0,Y 298.647,Z 538.096,A -85,B 0,C 180,E1 -16475.401,E2 -16475.401} C_VEL
LIN {X 0,Y 298.717,Z 538.087,A -85,B 0,C 180,E1 -16478.115,E2 -16478.115} C_VEL
LIN {X 0,Y 298.555,Z 538.107,A -85,B 0,C 180,E1 -16482.231,E2 -16482.231} C_VEL
LIN {X 0,Y 298.609,Z 538.099,A -85,B 0,C 180,E1 -16485.209,E2 -16485.209} C_VEL
LIN {X 0,Y 298.542,Z 538.106,A -85,B 0,C 180,E1 -16489.243,E2 -16489.243} C_VEL
LIN {X 0,Y 298.431,Z 538.123,A -85,B 0,C 180,E1 -16493.599,E2 -16493.599} C_VEL
LIN {X 0,Y 298.489,Z 538.114,A -85,B 0,C 180,E1 -16496.574,E2 -16496.574} C_VEL
LIN {X 0,Y 298.418,Z 538.124,A -85,B 0,C 180,E1 -16499.641,E2 -16499.641} C_VEL
LIN {X 0,Y 298.397,Z 538.125,A -85,B 0,C 180,E1 -16502.799,E2 -16502.799} C_VEL
LIN {X 0,Y 298.471,Z 538.115,A -85,B 0,C 180,E1 -16506.813,E2 -16506.813} C_VEL
LIN {X 0,Y 298.455,Z 538.117,A -85,B 0,C 180,E1 -16511.102,E2 -16511.102} C_VEL
LIN {X 0,Y 298.459,Z 538.117,A -85,B 0,C 180,E1 -16513.115,E2 -16513.115} C_VEL
LIN {X 0,Y 298.431,Z 538.12,A -85,B 0,C 180,E1 -16516.925,E2 -16516.925} C_VEL
LIN {X 0,Y 298.413,Z 538.123,A -85,B 0,C 180,E1 -16521.003,E2 -16521.003} C_VEL
LIN {X 0,Y 298.418,Z 538.125,A -85,B 0,C 180,E1 -16523.929,E2 -16523.929} C_VEL
LIN {X 0,Y 298.397,Z 538.128,A -85,B 0,C 180,E1 -16527.981,E2 -16527.981} C_VEL
LIN {X 0,Y 298.46,Z 538.119,A -85,B 0,C 180,E1 -16531.903,E2 -16531.903} C_VEL
LIN {X 0,Y 298.482,Z 538.115,A -85,B 0,C 180,E1 -16534.923,E2 -16534.923} C_VEL
LIN {X 0,Y 298.46,Z 538.117,A -85,B 0,C 180,E1 -16539.315,E2 -16539.315} C_VEL
LIN {X 0,Y 298.534,Z 538.111,A -85,B 0,C 180,E1 -16542.179,E2 -16542.179} C_VEL
LIN {X 0,Y 298.588,Z 538.102,A -85,B 0,C 180,E1 -16544.994,E2 -16544.994} C_VEL
LIN {X 0,Y 298.594,Z 538.099,A -85,B 0,C 180,E1 -16549.447,E2 -16549.447} C_VEL
LIN {X 0,Y 297.959,Z 538.182,A -85,B 0,C 180,E1 -16550.574,E2 -16550.574} C_VEL
LIN {X 0,Y 295.128,Z 538.536,A -85,B 0,C 180,E1 -16552.411,E2 -16552.411} C_VEL
LIN {X 0,Y 292.701,Z 538.837,A -85,B 0,C 180,E1 -16553.901,E2 -16553.901} C_VEL
LIN {X 0,Y 291.646,Z 538.967,A -85,B 0,C 180,E1 -16555.055,E2 -16555.055} C_VEL
LIN {X 0,Y 291.554,Z 538.977,A -85,B 0,C 180,E1 -16555.447,E2 -16555.447} C_VEL
LIN {X 0,Y 291.884,Z 538.939,A -85,B 0,C 180,E1 -16558.62,E2 -16558.62} C_VEL
LIN {X 0,Y 291.883,Z 538.936,A -85,B 0,C 180,E1 -16561.379,E2 -16561.379} C_VEL
LIN {X 0,Y 291.735,Z 538.956,A -85,B 0,C 180,E1 -16566.918,E2 -16566.918} C_VEL
LIN {X 0,Y 291.623,Z 538.968,A -85,B 0,C 180,E1 -16569.712,E2 -16569.712} C_VEL
LIN {X 0,Y 291.515,Z 538.983,A -85,B 0,C 180,E1 -16573.95,E2 -16573.95} C_VEL
LIN {X 0,Y 291.48,Z 538.989,A -85,B 0,C 180,E1 -16576.818,E2 -16576.818} C_VEL
LIN {X 0,Y 291.445,Z 538.99,A -85,B 0,C 180,E1 -16579.875,E2 -16579.875} C_VEL
LIN {X 0,Y 291.377,Z 539.001,A -85,B 0,C 180,E1 -16584.207,E2 -16584.207} C_VEL
LIN {X 0,Y 291.42,Z 538.994,A -85,B 0,C 180,E1 -16587.271,E2 -16587.271} C_VEL
LIN {X 0,Y 291.332,Z 539.007,A -85,B 0,C 180,E1 -16590.437,E2 -16590.437} C_VEL
LIN {X 0,Y 291.339,Z 539.004,A -85,B 0,C 180,E1 -16593.699,E2 -16593.699} C_VEL
LIN {X 0,Y 291.367,Z 539.002,A -85,B 0,C 180,E1 -16597.253,E2 -16597.253} C_VEL
LIN {X 0,Y 291.328,Z 539.009,A -85,B 0,C 180,E1 -16600.643,E2 -16600.643} C_VEL
LIN {X 0,Y 291.31,Z 539.009,A -85,B 0,C 180,E1 -16604.398,E2 -16604.398} C_VEL
LIN {X 0,Y 291.323,Z 539.008,A -85,B 0,C 180,E1 -16608.404,E2 -16608.404} C_VEL
LIN {X 0,Y 291.351,Z 539.006,A -85,B 0,C 180,E1 -16611.159,E2 -16611.159} C_VEL
LIN {X 0,Y 291.509,Z 539.2,A -85,B 0,C 180,E1 -16614.01,E2 -16614.01} C_VEL
LIN {X 0,Y 294.303,Z 553.522,A -85,B 0,C 180,E1 -16618.809,E2 -16618.809} C_VEL
LIN {X 0,Y 294.986,Z 557.16,A -85,B 0,C 180,E1 -16619.979,E2 -16619.979} C_VEL
LIN {X 0,Y 293.611,Z 568.089,A -85,B 0,C 180,E1 -16623.333,E2 -16623.333} C_VEL
LIN {X 0,Y 291.75,Z 584.826,A -85,B 0,C 180,E1 -16628.448,E2 -16628.448} C_VEL
LIN {X 0,Y 291.568,Z 587.328,A -85,B 0,C 180,E1 -16629.158,E2 -16629.158} C_VEL
LIN {X 0,Y 291.892,Z 594.667,A -85,B 0,C 180,E1 -16629.492,E2 -16629.492} C_VEL
LIN {X 0,Y 295.858,Z 651.448,A -85,B 0,C 180,E1 -16631.655,E2 -16631.655} C_VEL
LIN {X 0,Y 295.179,Z 674.298,A -85,B 0,C 180,E1 -16632.495,E2 -16632.495} C_VEL
LIN {X 0,Y 294.635,Z 686.193,A -85,B 0,C 180,E1 -16633.203,E2 -16633.203} C_VEL
LIN {X 0,Y 293.601,Z 698.112,A -85,B 0,C 180,E1 -16634.2,E2 -16634.2} C_VEL
LIN {X 0,Y 292.65,Z 708.789,A -85,B 0,C 180,E1 -16635.395,E2 -16635.395} C_VEL
LIN {X 0,Y 291.875,Z 718.405,A -85,B 0,C 180,E1 -16636.777,E2 -16636.777} C_VEL
LIN {X 0,Y 291.059,Z 727.918,A -85,B 0,C 180,E1 -16638.51,E2 -16638.51} C_VEL
LIN {X 0,Y 290.627,Z 735.476,A -85,B 0,C 180,E1 -16640.254,E2 -16640.254} C_VEL
LIN {X 0,Y 290.501,Z 741.989,A -85,B 0,C 180,E1 -16642.161,E2 -16642.161} C_VEL
LIN {X 0,Y 290.706,Z 747.903,A -85,B 0,C 180,E1 -16644.451,E2 -16644.451} C_VEL
LIN {X 0,Y 290.953,Z 751.654,A -85,B 0,C 180,E1 -16646.538,E2 -16646.538} C_VEL
LIN {X 0,Y 291.293,Z 754.052,A -85,B 0,C 180,E1 -16648.617,E2 -16648.617} C_VEL
LIN {X 0,Y 291.515,Z 754.894,A -85,B 0,C 180,E1 -16650,E2 -16650} C_VEL
LIN {X 0,Y 291.035,Z 755.107,A -85,B 0,C 180,E1 -16651.384,E2 -16651.384} C_VEL
LIN {X 0,Y 290.775,Z 754.773,A -85,B 0,C 180,E1 -16652.771,E2 -16652.771} C_VEL
LIN {X 0,Y 290.525,Z 753.938,A -85,B 0,C 180,E1 -16654.162,E2 -16654.162} C_VEL
LIN {X 0,Y 290.121,Z 751.019,A -85,B 0,C 180,E1 -16656.689,E2 -16656.689} C_VEL
LIN {X 0,Y 290.208,Z 746.693,A -85,B 0,C 180,E1 -16659.056,E2 -16659.056} C_VEL
LIN {X 0,Y 290.664,Z 741.467,A -85,B 0,C 180,E1 -16661.153,E2 -16661.153} C_VEL
LIN {X 0,Y 291.423,Z 735.972,A -85,B 0,C 180,E1 -16662.889,E2 -16662.889} C_VEL
LIN {X 0,Y 293.016,Z 727.723,A -85,B 0,C 180,E1 -16664.941,E2 -16664.941} C_VEL
LIN {X 0,Y 294.633,Z 719.154,A -85,B 0,C 180,E1 -16666.633,E2 -16666.633} C_VEL
LIN {X 0,Y 296.797,Z 708.55,A -85,B 0,C 180,E1 -16668.285,E2 -16668.285} C_VEL
LIN {X 0,Y 298.872,Z 697.246,A -85,B 0,C 180,E1 -16669.654,E2 -16669.654} C_VEL
LIN {X 0,Y 300.727,Z 685.993,A -85,B 0,C 180,E1 -16670.699,E2 -16670.699} C_VEL
LIN {X 0,Y 302.332,Z 673.645,A -85,B 0,C 180,E1 -16671.566,E2 -16671.566} C_VEL
LIN {X 0,Y 303.579,Z 659.979,A -85,B 0,C 180,E1 -16672.227,E2 -16672.227} C_VEL
LIN {X 0,Y 303.808,Z 651.169,A -85,B 0,C 180,E1 -16672.55,E2 -16672.55} C_VEL
LIN {X 0,Y 303.151,Z 627.767,A -85,B 0,C 180,E1 -16673.538,E2 -16673.538} C_VEL
LIN {X 0,Y 301.539,Z 610.633,A -85,B 0,C 180,E1 -16674.436,E2 -16674.436} C_VEL
LIN {X 0,Y 299.137,Z 594.025,A -85,B 0,C 180,E1 -16675.452,E2 -16675.452} C_VEL
LIN {X 0,Y 295.849,Z 577.278,A -85,B 0,C 180,E1 -16676.67,E2 -16676.67} C_VEL
LIN {X 0,Y 293.936,Z 568.198,A -85,B 0,C 180,E1 -16677.437,E2 -16677.437} C_VEL
LIN {X 0,Y 294.789,Z 562.182,A -85,B 0,C 180,E1 -16679.257,E2 -16679.257} C_VEL
LIN {X 0,Y 295.19,Z 558.499,A -85,B 0,C 180,E1 -16680.47,E2 -16680.47} C_VEL
LIN {X 0,Y 293.873,Z 550.62,A -85,B 0,C 180,E1 -16683.369,E2 -16683.369} C_VEL
LIN {X 0,Y 292.277,Z 542.799,A -85,B 0,C 180,E1 -16686.52,E2 -16686.52} C_VEL
LIN {X 0,Y 291.378,Z 539.057,A -85,B 0,C 180,E1 -16688.221,E2 -16688.221} C_VEL
LIN {X 0,Y 291.335,Z 539.004,A -85,B 0,C 180,E1 -16692.488,E2 -16692.488} C_VEL
LIN {X 0,Y 291.366,Z 539.005,A -85,B 0,C 180,E1 -16696.353,E2 -16696.353} C_VEL
LIN {X 0,Y 291.408,Z 538.993,A -85,B 0,C 180,E1 -16700.51,E2 -16700.51} C_VEL
LIN {X 0,Y 291.429,Z 538.996,A -85,B 0,C 180,E1 -16702.923,E2 -16702.923} C_VEL
LIN {X 0,Y 291.34,Z 539.007,A -85,B 0,C 180,E1 -16706.302,E2 -16706.302} C_VEL
LIN {X 0,Y 291.382,Z 538.995,A -85,B 0,C 180,E1 -16710.26,E2 -16710.26} C_VEL
LIN {X 0,Y 291.41,Z 538.992,A -85,B 0,C 180,E1 -16714.272,E2 -16714.272} C_VEL
LIN {X 0,Y 291.382,Z 538.997,A -85,B 0,C 180,E1 -16717.3,E2 -16717.3} C_VEL
LIN {X 0,Y 291.451,Z 538.989,A -85,B 0,C 180,E1 -16720.27,E2 -16720.27} C_VEL
LIN {X 0,Y 291.534,Z 538.979,A -85,B 0,C 180,E1 -16724.635,E2 -16724.635} C_VEL
LIN {X 0,Y 291.531,Z 538.982,A -85,B 0,C 180,E1 -16728.881,E2 -16728.881} C_VEL
LIN {X 0,Y 291.743,Z 539.113,A -85,B 0,C 180,E1 -16731.951,E2 -16731.951} C_VEL
LIN {X 0,Y 291.958,Z 540.095,A -85,B 0,C 180,E1 -16732.262,E2 -16732.262} C_VEL
LIN {X 0,Y 293.613,Z 542.944,A -85,B 0,C 180,E1 -16732.688,E2 -16732.688} C_VEL
LIN {X 0,Y 294.747,Z 544.471,A -85,B 0,C 180,E1 -16732.943,E2 -16732.943} C_VEL
LIN {X 0,Y 304.482,Z 561.148,A -85,B 0,C 180,E1 -16735.093,E2 -16735.093} C_VEL
LIN {X 0,Y 308.119,Z 568.67,A -85,B 0,C 180,E1 -16735.863,E2 -16735.863} C_VEL
LIN {X 0,Y 307.932,Z 585.978,A -85,B 0,C 180,E1 -16736.493,E2 -16736.493} C_VEL
LIN {X 0,Y 307.543,Z 597.658,A -85,B 0,C 180,E1 -16737.166,E2 -16737.166} C_VEL
LIN {X 0,Y 306.721,Z 608.702,A -85,B 0,C 180,E1 -16738.031,E2 -16738.031} C_VEL
LIN {X 0,Y 305.458,Z 620.009,A -85,B 0,C 180,E1 -16739.177,E2 -16739.177} C_VEL
LIN {X 0,Y 304.044,Z 630.108,A -85,B 0,C 180,E1 -16740.497,E2 -16740.497} C_VEL
LIN {X 0,Y 302.396,Z 639.742,A -85,B 0,C 180,E1 -16742.082,E2 -16742.082} C_VEL
LIN {X 0,Y 300.771,Z 647.672,A -85,B 0,C 180,E1 -16743.685,E2 -16743.685} C_VEL
LIN {X 0,Y 298.929,Z 655.673,A -85,B 0,C 180,E1 -16745.735,E2 -16745.735} C_VEL
LIN {X 0,Y 297.426,Z 661.367,A -85,B 0,C 180,E1 -16747.583,E2 -16747.583} C_VEL
LIN {X 0,Y 296.027,Z 666.15,A -85,B 0,C 180,E1 -16749.567,E2 -16749.567} C_VEL
LIN {X 0,Y 294.581,Z 670.409,A -85,B 0,C 180,E1 -16752.003,E2 -16752.003} C_VEL
LIN {X 0,Y 293.697,Z 672.609,A -85,B 0,C 180,E1 -16753.845,E2 -16753.845} C_VEL
LIN {X 0,Y 292.8,Z 674.241,A -85,B 0,C 180,E1 -16756.243,E2 -16756.243} C_VEL
LIN {X 0,Y 292.236,Z 674.61,A -85,B 0,C 180,E1 -16758.219,E2 -16758.219} C_VEL
LIN {X 0,Y 291.894,Z 674.133,A -85,B 0,C 180,E1 -16760.118,E2 -16760.118} C_VEL
LIN {X 0,Y 291.665,Z 672.21,A -85,B 0,C 180,E1 -16762.678,E2 -16762.678} C_VEL
LIN {X 0,Y 291.742,Z 669.271,A -85,B 0,C 180,E1 -16764.934,E2 -16764.934} C_VEL
LIN {X 0,Y 292.043,Z 664.999,A -85,B 0,C 180,E1 -16767.209,E2 -16767.209} C_VEL
LIN {X 0,Y 292.486,Z 659.403,A -85,B 0,C 180,E1 -16769.457,E2 -16769.457} C_VEL
LIN {X 0,Y 293.052,Z 653.132,A -85,B 0,C 180,E1 -16771.441,E2 -16771.441} C_VEL
LIN {X 0,Y 293.752,Z 645.466,A -85,B 0,C 180,E1 -16773.386,E2 -16773.386} C_VEL
LIN {X 0,Y 294.629,Z 636.376,A -85,B 0,C 180,E1 -16775.252,E2 -16775.252} C_VEL
LIN {X 0,Y 295.463,Z 626.343,A -85,B 0,C 180,E1 -16776.914,E2 -16776.914} C_VEL
LIN {X 0,Y 296.216,Z 615.396,A -85,B 0,C 180,E1 -16778.364,E2 -16778.364} C_VEL
LIN {X 0,Y 297.009,Z 603.412,A -85,B 0,C 180,E1 -16779.608,E2 -16779.608} C_VEL
LIN {X 0,Y 297.583,Z 590.994,A -85,B 0,C 180,E1 -16780.582,E2 -16780.582} C_VEL
LIN {X 0,Y 297.829,Z 578.367,A -85,B 0,C 180,E1 -16781.297,E2 -16781.297} C_VEL
LIN {X 0,Y 297.924,Z 559.623,A -85,B 0,C 180,E1 -16781.941,E2 -16781.941} C_VEL
LIN {X 0,Y 291.561,Z 540.017,A -85,B 0,C 180,E1 -16782.869,E2 -16782.869} C_VEL
LIN {X 0,Y 291.4,Z 539.124,A -85,B 0,C 180,E1 -16783.109,E2 -16783.109} C_VEL
LIN {X 0,Y 291.397,Z 539.002,A -85,B 0,C 180,E1 -16787.523,E2 -16787.523} C_VEL
LIN {X 0,Y 291.385,Z 539.002,A -85,B 0,C 180,E1 -16791.165,E2 -16791.165} C_VEL
LIN {X 0,Y 291.386,Z 538.998,A -85,B 0,C 180,E1 -16794.631,E2 -16794.631} C_VEL
LIN {X 0,Y 291.373,Z 539.001,A -85,B 0,C 180,E1 -16797.952,E2 -16797.952} C_VEL
LIN {X 0,Y 291.384,Z 539.001,A -85,B 0,C 180,E1 -16801.159,E2 -16801.159} C_VEL
LIN {X 0,Y 291.419,Z 538.994,A -85,B 0,C 180,E1 -16804.273,E2 -16804.273} C_VEL
LIN {X 0,Y 291.382,Z 539.001,A -85,B 0,C 180,E1 -16807.3,E2 -16807.3} C_VEL
LIN {X 0,Y 291.461,Z 538.989,A -85,B 0,C 180,E1 -16810.271,E2 -16810.271} C_VEL
LIN {X 0,Y 291.518,Z 538.981,A -85,B 0,C 180,E1 -16814.654,E2 -16814.654} C_VEL
LIN {X 0,Y 291.539,Z 538.979,A -85,B 0,C 180,E1 -16818.881,E2 -16818.881} C_VEL
LIN {X 0,Y 291.668,Z 538.967,A -85,B 0,C 180,E1 -16821.688,E2 -16821.688} C_VEL
LIN {X 0,Y 291.616,Z 538.969,A -85,B 0,C 180,E1 -16824.468,E2 -16824.468} C_VEL
LIN {X 0,Y 291.893,Z 538.935,A -85,B 0,C 180,E1 -16828.62,E2 -16828.62} C_VEL
LIN {X 0,Y 291.893,Z 538.936,A -85,B 0,C 180,E1 -16831.38,E2 -16831.38} C_VEL
LIN {X 0,Y 291.616,Z 538.972,A -85,B 0,C 180,E1 -16835.532,E2 -16835.532} C_VEL
LIN {X 0,Y 291.678,Z 538.961,A -85,B 0,C 180,E1 -16838.919,E2 -16838.919} C_VEL
LIN {X 0,Y 291.526,Z 538.985,A -85,B 0,C 180,E1 -16843.95,E2 -16843.95} C_VEL
LIN {X 0,Y 291.491,Z 538.985,A -85,B 0,C 180,E1 -16846.817,E2 -16846.817} C_VEL
LIN {X 0,Y 291.454,Z 538.994,A -85,B 0,C 180,E1 -16849.874,E2 -16849.874} C_VEL
LIN {X 0,Y 291.386,Z 539.001,A -85,B 0,C 180,E1 -16854.206,E2 -16854.206} C_VEL
LIN {X 0,Y 291.422,Z 538.993,A -85,B 0,C 180,E1 -16857.271,E2 -16857.271} C_VEL
LIN {X 0,Y 291.336,Z 539.006,A -85,B 0,C 180,E1 -16860.436,E2 -16860.436} C_VEL
LIN {X 0,Y 291.346,Z 539.006,A -85,B 0,C 180,E1 -16863.697,E2 -16863.697} C_VEL
LIN {X 0,Y 291.405,Z 538.995,A -85,B 0,C 180,E1 -16867.26,E2 -16867.26} C_VEL
LIN {X 0,Y 291.406,Z 538.997,A -85,B 0,C 180,E1 -16870.629,E2 -16870.629} C_VEL
LIN {X 0,Y 291.353,Z 539.004,A -85,B 0,C 180,E1 -16874.389,E2 -16874.389} C_VEL
LIN {X 0,Y 291.33,Z 539.008,A -85,B 0,C 180,E1 -16878.402,E2 -16878.402} C_VEL
LIN {X 0,Y 291.362,Z 539.001,A -85,B 0,C 180,E1 -16881.159,E2 -16881.159} C_VEL
LIN {X 0,Y 291.36,Z 539.002,A -85,B 0,C 180,E1 -16884.625,E2 -16884.625} C_VEL
LIN {X 0,Y 291.373,Z 539.003,A -85,B 0,C 180,E1 -16887.95,E2 -16887.95} C_VEL
LIN {X 0,Y 291.379,Z 538.999,A -85,B 0,C 180,E1 -16891.157,E2 -16891.157} C_VEL
LIN {X 0,Y 291.414,Z 538.999,A -85,B 0,C 180,E1 -16894.271,E2 -16894.271} C_VEL
LIN {X 0,Y 291.386,Z 538.998,A -85,B 0,C 180,E1 -16897.299,E2 -16897.299} C_VEL
LIN {X 0,Y 291.459,Z 538.994,A -85,B 0,C 180,E1 -16900.27,E2 -16900.27} C_VEL
LIN {X 0,Y 291.536,Z 538.982,A -85,B 0,C 180,E1 -16904.634,E2 -16904.634} C_VEL
LIN {X 0,Y 291.533,Z 538.981,A -85,B 0,C 180,E1 -16908.88,E2 -16908.88} C_VEL
LIN {X 0,Y 291.703,Z 538.958,A -85,B 0,C 180,E1 -16911.688,E2 -16911.688} C_VEL
LIN {X 0,Y 291.626,Z 538.974,A -85,B 0,C 180,E1 -16914.468,E2 -16914.468} C_VEL
LIN {X 0,Y 291.554,Z 538.977,A -85,B 0,C 180,E1 -16915.447,E2 -16915.447} C_VEL
LIN {X 0,Y 290.924,Z 539.06,A -85,B 0,C 180,E1 -16916.602,E2 -16916.602} C_VEL
LIN {X 0,Y 288.274,Z 539.39,A -85,B 0,C 180,E1 -16918.489,E2 -16918.489} C_VEL
LIN {X 0,Y 285.192,Z 539.772,A -85,B 0,C 180,E1 -16920.804,E2 -16920.804} C_VEL
LIN {X 0,Y 284.825,Z 539.814,A -85,B 0,C 180,E1 -16921.601,E2 -16921.601} C_VEL
LIN {X 0,Y 284.688,Z 539.833,A -85,B 0,C 180,E1 -16927.09,E2 -16927.09} C_VEL
LIN {X 0,Y 284.56,Z 539.848,A -85,B 0,C 180,E1 -16929.955,E2 -16929.955} C_VEL
LIN {X 0,Y 284.472,Z 539.862,A -85,B 0,C 180,E1 -16934.303,E2 -16934.303} C_VEL
LIN {X 0,Y 284.417,Z 539.866,A -85,B 0,C 180,E1 -16937.248,E2 -16937.248} C_VEL
LIN {X 0,Y 284.371,Z 539.873,A -85,B 0,C 180,E1 -16940.242,E2 -16940.242} C_VEL
LIN {X 0,Y 284.334,Z 539.88,A -85,B 0,C 180,E1 -16944.846,E2 -16944.846} C_VEL
LIN {X 0,Y 284.329,Z 539.877,A -85,B 0,C 180,E1 -16948.01,E2 -16948.01} C_VEL
LIN {X 0,Y 284.29,Z 539.883,A -85,B 0,C 180,E1 -16951.274,E2 -16951.274} C_VEL
LIN {X 0,Y 284.336,Z 539.876,A -85,B 0,C 180,E1 -16955.348,E2 -16955.348} C_VEL
LIN {X 0,Y 284.303,Z 539.881,A -85,B 0,C 180,E1 -16958.17,E2 -16958.17} C_VEL
LIN {X 0,Y 284.265,Z 539.886,A -85,B 0,C 180,E1 -16962.125,E2 -16962.125} C_VEL
LIN {X 0,Y 284.264,Z 539.886,A -85,B 0,C 180,E1 -16966.192,E2 -16966.192} C_VEL
LIN {X 0,Y 284.303,Z 539.881,A -85,B 0,C 180,E1 -16970.024,E2 -16970.024} C_VEL
LIN {X 0,Y 284.468,Z 539.931,A -85,B 0,C 180,E1 -16973.77,E2 -16973.77} C_VEL
LIN {X 0,Y 286.62,Z 551.288,A -85,B 0,C 180,E1 -16977.752,E2 -16977.752} C_VEL
LIN {X 0,Y 287.915,Z 557.972,A -85,B 0,C 180,E1 -16979.974,E2 -16979.974} C_VEL
LIN {X 0,Y 286.317,Z 570.022,A -85,B 0,C 180,E1 -16983.78,E2 -16983.78} C_VEL
LIN {X 0,Y 284.594,Z 585.863,A -85,B 0,C 180,E1 -16988.729,E2 -16988.729} C_VEL
LIN {X 0,Y 284.566,Z 587.662,A -85,B 0,C 180,E1 -16988.891,E2 -16988.891} C_VEL
LIN {X 0,Y 288.868,Z 651.94,A -85,B 0,C 180,E1 -16991.424,E2 -16991.424} C_VEL
LIN {X 0,Y 288.209,Z 673.744,A -85,B 0,C 180,E1 -16992.261,E2 -16992.261} C_VEL
LIN {X 0,Y 287.604,Z 686.141,A -85,B 0,C 180,E1 -16993.04,E2 -16993.04} C_VEL
LIN {X 0,Y 286.634,Z 697.032,A -85,B 0,C 180,E1 -16993.988,E2 -16993.988} C_VEL
LIN {X 0,Y 285.632,Z 707.672,A -85,B 0,C 180,E1 -16995.21,E2 -16995.21} C_VEL
LIN {X 0,Y 284.851,Z 717.294,A -85,B 0,C 180,E1 -16996.626,E2 -16996.626} C_VEL
LIN {X 0,Y 284.072,Z 725.967,A -85,B 0,C 180,E1 -16998.223,E2 -16998.223} C_VEL
LIN {X 0,Y 283.619,Z 733.677,A -85,B 0,C 180,E1 -17000.011,E2 -17000.011} C_VEL
LIN {X 0,Y 283.475,Z 739.993,A -85,B 0,C 180,E1 -17001.84,E2 -17001.84} C_VEL
LIN {X 0,Y 283.556,Z 744.788,A -85,B 0,C 180,E1 -17003.596,E2 -17003.596} C_VEL
LIN {X 0,Y 283.857,Z 749.179,A -85,B 0,C 180,E1 -17005.74,E2 -17005.74} C_VEL
LIN {X 0,Y 284.004,Z 751.298,A -85,B 0,C 180,E1 -17007.163,E2 -17007.163} C_VEL
LIN {X 0,Y 284.271,Z 752.81,A -85,B 0,C 180,E1 -17008.583,E2 -17008.583} C_VEL
LIN {X 0,Y 284.49,Z 753.743,A -85,B 0,C 180,E1 -17010,E2 -17010} C_VEL
LIN {X 0,Y 284.002,Z 754.002,A -85,B 0,C 180,E1 -17011.418,E2 -17011.418} C_VEL
LIN {X 0,Y 283.714,Z 753.749,A -85,B 0,C 180,E1 -17012.84,E2 -17012.84} C_VEL
LIN {X 0,Y 283.449,Z 752.956,A -85,B 0,C 180,E1 -17014.266,E2 -17014.266} C_VEL
LIN {X 0,Y 283.057,Z 750.378,A -85,B 0,C 180,E1 -17016.71,E2 -17016.71} C_VEL
LIN {X 0,Y 283.14,Z 746.016,A -85,B 0,C 180,E1 -17019.284,E2 -17019.284} C_VEL
LIN {X 0,Y 283.759,Z 739.926,A -85,B 0,C 180,E1 -17021.79,E2 -17021.79} C_VEL
LIN {X 0,Y 284.993,Z 733.056,A -85,B 0,C 180,E1 -17023.912,E2 -17023.912} C_VEL
LIN {X 0,Y 286.446,Z 726.016,A -85,B 0,C 180,E1 -17025.657,E2 -17025.657} C_VEL
LIN {X 0,Y 288.222,Z 717.386,A -85,B 0,C 180,E1 -17027.379,E2 -17027.379} C_VEL
LIN {X 0,Y 290.353,Z 707.84,A -85,B 0,C 180,E1 -17028.889,E2 -17028.889} C_VEL
LIN {X 0,Y 292.387,Z 697.395,A -85,B 0,C 180,E1 -17030.203,E2 -17030.203} C_VEL
LIN {X 0,Y 294.432,Z 685.676,A -85,B 0,C 180,E1 -17031.346,E2 -17031.346} C_VEL
LIN {X 0,Y 296.3,Z 672.479,A -85,B 0,C 180,E1 -17032.303,E2 -17032.303} C_VEL
LIN {X 0,Y 297.611,Z 659.102,A -85,B 0,C 180,E1 -17032.977,E2 -17032.977} C_VEL
LIN {X 0,Y 297.819,Z 650.33,A -85,B 0,C 180,E1 -17033.328,E2 -17033.328} C_VEL
LIN {X 0,Y 297.231,Z 628.216,A -85,B 0,C 180,E1 -17034.302,E2 -17034.302} C_VEL
LIN {X 0,Y 295.799,Z 612.456,A -85,B 0,C 180,E1 -17035.153,E2 -17035.153} C_VEL
LIN {X 0,Y 293.586,Z 596.137,A -85,B 0,C 180,E1 -17036.198,E2 -17036.198} C_VEL
LIN {X 0,Y 290.502,Z 580.031,A -85,B 0,C 180,E1 -17037.415,E2 -17037.415} C_VEL
LIN {X 0,Y 288.057,Z 569.354,A -85,B 0,C 180,E1 -17038.345,E2 -17038.345} C_VEL
LIN {X 0,Y 287.489,Z 565.805,A -85,B 0,C 180,E1 -17038.696,E2 -17038.696} C_VEL
LIN {X 0,Y 288.242,Z 560.501,A -85,B 0,C 180,E1 -17040.392,E2 -17040.392} C_VEL
LIN {X 0,Y 287.477,Z 554.71,A -85,B 0,C 180,E1 -17042.536,E2 -17042.536} C_VEL
LIN {X 0,Y 285.884,Z 546.687,A -85,B 0,C 180,E1 -17045.782,E2 -17045.782} C_VEL
LIN {X 0,Y 284.335,Z 539.951,A -85,B 0,C 180,E1 -17048.843,E2 -17048.843} C_VEL
LIN {X 0,Y 284.278,Z 539.883,A -85,B 0,C 180,E1 -17052.127,E2 -17052.127} C_VEL
LIN {X 0,Y 284.314,Z 539.883,A -85,B 0,C 180,E1 -17056.201,E2 -17056.201} C_VEL
LIN {X 0,Y 284.346,Z 539.876,A -85,B 0,C 180,E1 -17060.013,E2 -17060.013} C_VEL
LIN {X 0,Y 284.35,Z 539.871,A -85,B 0,C 180,E1 -17063.617,E2 -17063.617} C_VEL
LIN {X 0,Y 284.303,Z 539.876,A -85,B 0,C 180,E1 -17067.189,E2 -17067.189} C_VEL
LIN {X 0,Y 284.353,Z 539.87,A -85,B 0,C 180,E1 -17070.376,E2 -17070.376} C_VEL
LIN {X 0,Y 284.371,Z 539.867,A -85,B 0,C 180,E1 -17073.586,E2 -17073.586} C_VEL
LIN {X 0,Y 284.362,Z 539.87,A -85,B 0,C 180,E1 -17076.707,E2 -17076.707} C_VEL
LIN {X 0,Y 284.397,Z 539.872,A -85,B 0,C 180,E1 -17081.262,E2 -17081.262} C_VEL
LIN {X 0,Y 284.471,Z 539.859,A -85,B 0,C 180,E1 -17084.47,E2 -17084.47} C_VEL
LIN {X 0,Y 284.483,Z 539.861,A -85,B 0,C 180,E1 -17088.602,E2 -17088.602} C_VEL
LIN {X 0,Y 284.666,Z 540.072,A -85,B 0,C 180,E1 -17090.679,E2 -17090.679} C_VEL
LIN {X 0,Y 284.95,Z 541.158,A -85,B 0,C 180,E1 -17090.984,E2 -17090.984} C_VEL
LIN {X 0,Y 286.538,Z 543.823,A -85,B 0,C 180,E1 -17091.426,E2 -17091.426} C_VEL
LIN {X 0,Y 287.715,Z 545.216,A -85,B 0,C 180,E1 -17091.716,E2 -17091.716} C_VEL
LIN {X 0,Y 289.866,Z 548.572,A -85,B 0,C 180,E1 -17092.266,E2 -17092.266} C_VEL
LIN {X 0,Y 299.561,Z 565.296,A -85,B 0,C 180,E1 -17094.525,E2 -17094.525} C_VEL
LIN {X 0,Y 302.393,Z 571.352,A -85,B 0,C 180,E1 -17095.158,E2 -17095.158} C_VEL
LIN {X 0,Y 302.136,Z 587.672,A -85,B 0,C 180,E1 -17095.781,E2 -17095.781} C_VEL
LIN {X 0,Y 301.687,Z 598.784,A -85,B 0,C 180,E1 -17096.441,E2 -17096.441} C_VEL
LIN {X 0,Y 300.803,Z 609.788,A -85,B 0,C 180,E1 -17097.322,E2 -17097.322} C_VEL
LIN {X 0,Y 299.467,Z 621.12,A -85,B 0,C 180,E1 -17098.488,E2 -17098.488} C_VEL
LIN {X 0,Y 297.982,Z 631.257,A -85,B 0,C 180,E1 -17099.832,E2 -17099.832} C_VEL
LIN {X 0,Y 296.282,Z 640.483,A -85,B 0,C 180,E1 -17101.36,E2 -17101.36} C_VEL
LIN {X 0,Y 294.475,Z 648.845,A -85,B 0,C 180,E1 -17103.079,E2 -17103.079} C_VEL
LIN {X 0,Y 292.493,Z 656.814,A -85,B 0,C 180,E1 -17105.17,E2 -17105.17} C_VEL
LIN {X 0,Y 290.596,Z 663.551,A -85,B 0,C 180,E1 -17107.453,E2 -17107.453} C_VEL
LIN {X 0,Y 288.901,Z 668.69,A -85,B 0,C 180,E1 -17109.805,E2 -17109.805} C_VEL
LIN {X 0,Y 287.552,Z 672.322,A -85,B 0,C 180,E1 -17112.148,E2 -17112.148} C_VEL
LIN {X 0,Y 286.562,Z 674.385,A -85,B 0,C 180,E1 -17114.197,E2 -17114.197} C_VEL
LIN {X 0,Y 285.749,Z 675.555,A -85,B 0,C 180,E1 -17116.427,E2 -17116.427} C_VEL
LIN {X 0,Y 285.126,Z 675.633,A -85,B 0,C 180,E1 -17118.69,E2 -17118.69} C_VEL
LIN {X 0,Y 284.847,Z 674.986,A -85,B 0,C 180,E1 -17120.356,E2 -17120.356} C_VEL
LIN {X 0,Y 284.671,Z 674.03,A -85,B 0,C 180,E1 -17121.736,E2 -17121.736} C_VEL
LIN {X 0,Y 284.641,Z 671.512,A -85,B 0,C 180,E1 -17124.002,E2 -17124.002} C_VEL
LIN {X 0,Y 284.862,Z 667.63,A -85,B 0,C 180,E1 -17126.366,E2 -17126.366} C_VEL
LIN {X 0,Y 285.228,Z 662.402,A -85,B 0,C 180,E1 -17128.717,E2 -17128.717} C_VEL
LIN {X 0,Y 285.849,Z 655.453,A -85,B 0,C 180,E1 -17131.086,E2 -17131.086} C_VEL
LIN {X 0,Y 286.582,Z 647.958,A -85,B 0,C 180,E1 -17133.115,E2 -17133.115} C_VEL
LIN {X 0,Y 287.43,Z 638.937,A -85,B 0,C 180,E1 -17135.073,E2 -17135.073} C_VEL
LIN {X 0,Y 288.32,Z 628.642,A -85,B 0,C 180,E1 -17136.873,E2 -17136.873} C_VEL
LIN {X 0,Y 289.129,Z 618.398,A -85,B 0,C 180,E1 -17138.305,E2 -17138.305} C_VEL
LIN {X 0,Y 289.885,Z 606.411,A -85,B 0,C 180,E1 -17139.638,E2 -17139.638} C_VEL
LIN {X 0,Y 290.548,Z 594.283,A -85,B 0,C 180,E1 -17140.662,E2 -17140.662} C_VEL
LIN {X 0,Y 290.896,Z 581.317,A -85,B 0,C 180,E1 -17141.458,E2 -17141.458} C_VEL
LIN {X 0,Y 290.978,Z 568.041,A -85,B 0,C 180,E1 -17141.988,E2 -17141.988} C_VEL
LIN {X 0,Y 290.891,Z 560.625,A -85,B 0,C 180,E1 -17142.229,E2 -17142.229} C_VEL
LIN {X 0,Y 284.518,Z 540.818,A -85,B 0,C 180,E1 -17143.192,E2 -17143.192} C_VEL
LIN {X 0,Y 284.336,Z 539.944,A -85,B 0,C 180,E1 -17143.486,E2 -17143.486} C_VEL
LIN {X 0,Y 284.34,Z 539.878,A -85,B 0,C 180,E1 -17147.861,E2 -17147.861} C_VEL
LIN {X 0,Y 284.336,Z 539.879,A -85,B 0,C 180,E1 -17151.836,E2 -17151.836} C_VEL
LIN {X 0,Y 284.325,Z 539.883,A -85,B 0,C 180,E1 -17155.354,E2 -17155.354} C_VEL
LIN {X 0,Y 284.297,Z 539.882,A -85,B 0,C 180,E1 -17158.727,E2 -17158.727} C_VEL
LIN {X 0,Y 284.399,Z 539.869,A -85,B 0,C 180,E1 -17162.827,E2 -17162.827} C_VEL
LIN {X 0,Y 284.368,Z 539.872,A -85,B 0,C 180,E1 -17166.708,E2 -17166.708} C_VEL
LIN {X 0,Y 284.384,Z 539.873,A -85,B 0,C 180,E1 -17171.261,E2 -17171.261} C_VEL
LIN {X 0,Y 284.471,Z 539.864,A -85,B 0,C 180,E1 -17175.697,E2 -17175.697} C_VEL
LIN {X 0,Y 284.521,Z 539.855,A -85,B 0,C 180,E1 -17180.043,E2 -17180.043} C_VEL
LIN {X 0,Y 284.657,Z 539.835,A -85,B 0,C 180,E1 -17182.909,E2 -17182.909} C_VEL
LIN {X 0,Y 284.859,Z 539.811,A -85,B 0,C 180,E1 -17188.586,E2 -17188.586} C_VEL
LIN {X 0,Y 284.859,Z 539.813,A -85,B 0,C 180,E1 -17191.414,E2 -17191.414} C_VEL
LIN {X 0,Y 284.657,Z 539.837,A -85,B 0,C 180,E1 -17197.091,E2 -17197.091} C_VEL
LIN {X 0,Y 284.518,Z 539.857,A -85,B 0,C 180,E1 -17199.957,E2 -17199.957} C_VEL
LIN {X 0,Y 284.486,Z 539.859,A -85,B 0,C 180,E1 -17204.302,E2 -17204.302} C_VEL
LIN {X 0,Y 284.429,Z 539.865,A -85,B 0,C 180,E1 -17207.248,E2 -17207.248} C_VEL
LIN {X 0,Y 284.381,Z 539.873,A -85,B 0,C 180,E1 -17210.242,E2 -17210.242} C_VEL
LIN {X 0,Y 284.34,Z 539.876,A -85,B 0,C 180,E1 -17214.846,E2 -17214.846} C_VEL
LIN {X 0,Y 284.331,Z 539.881,A -85,B 0,C 180,E1 -17218.01,E2 -17218.01} C_VEL
LIN {X 0,Y 284.296,Z 539.882,A -85,B 0,C 180,E1 -17221.274,E2 -17221.274} C_VEL
LIN {X 0,Y 284.363,Z 539.873,A -85,B 0,C 180,E1 -17225.353,E2 -17225.353} C_VEL
LIN {X 0,Y 284.338,Z 539.88,A -85,B 0,C 180,E1 -17228.164,E2 -17228.164} C_VEL
LIN {X 0,Y 284.343,Z 539.88,A -85,B 0,C 180,E1 -17232.14,E2 -17232.14} C_VEL
LIN {X 0,Y 284.297,Z 539.885,A -85,B 0,C 180,E1 -17236.196,E2 -17236.196} C_VEL
LIN {X 0,Y 284.306,Z 539.884,A -85,B 0,C 180,E1 -17240.023,E2 -17240.023} C_VEL
LIN {X 0,Y 284.334,Z 539.877,A -85,B 0,C 180,E1 -17243.614,E2 -17243.614} C_VEL
LIN {X 0,Y 284.307,Z 539.88,A -85,B 0,C 180,E1 -17247.188,E2 -17247.188} C_VEL
LIN {X 0,Y 284.357,Z 539.878,A -85,B 0,C 180,E1 -17250.375,E2 -17250.375} C_VEL
LIN {X 0,Y 284.375,Z 539.871,A -85,B 0,C 180,E1 -17253.586,E2 -17253.586} C_VEL
LIN {X 0,Y 284.365,Z 539.875,A -85,B 0,C 180,E1 -17256.706,E2 -17256.706} C_VEL
LIN {X 0,Y 284.401,Z 539.867,A -85,B 0,C 180,E1 -17261.261,E2 -17261.261} C_VEL
LIN {X 0,Y 284.474,Z 539.863,A -85,B 0,C 180,E1 -17264.469,E2 -17264.469} C_VEL
LIN {X 0,Y 284.484,Z 539.861,A -85,B 0,C 180,E1 -17268.601,E2 -17268.601} C_VEL
LIN {X 0,Y 284.654,Z 539.835,A -85,B 0,C 180,E1 -17271.48,E2 -17271.48} C_VEL
LIN {X 0,Y 284.596,Z 539.848,A -85,B 0,C 180,E1 -17274.331,E2 -17274.331} C_VEL
LIN {X 0,Y 284.85,Z 539.816,A -85,B 0,C 180,E1 -17278.586,E2 -17278.586} C_VEL
LIN {X 0,Y 284.825,Z 539.814,A -85,B 0,C 180,E1 -17281.601,E2 -17281.601} C_VEL
LIN {X 0,Y 284.059,Z 539.914,A -85,B 0,C 180,E1 -17282.779,E2 -17282.779} C_VEL
LIN {X 0,Y 281.157,Z 540.276,A -85,B 0,C 180,E1 -17284.697,E2 -17284.697} C_VEL
LIN {X 0,Y 278.743,Z 540.576,A -85,B 0,C 180,E1 -17286.255,E2 -17286.255} C_VEL
LIN {X 0,Y 277.7,Z 540.703,A -85,B 0,C 180,E1 -17287.462,E2 -17287.462} C_VEL
LIN {X 0,Y 277.607,Z 540.713,A -85,B 0,C 180,E1 -17287.872,E2 -17287.872} C_VEL
LIN {X 0,Y 277.501,Z 540.729,A -85,B 0,C 180,E1 -17290.211,E2 -17290.211} C_VEL
LIN {X 0,Y 277.422,Z 540.742,A -85,B 0,C 180,E1 -17294.674,E2 -17294.674} C_VEL
LIN {X 0,Y 277.337,Z 540.748,A -85,B 0,C 180,E1 -17299.234,E2 -17299.234} C_VEL
LIN {X 0,Y 277.287,Z 540.756,A -85,B 0,C 180,E1 -17304.158,E2 -17304.158} C_VEL
LIN {X 0,Y 277.323,Z 540.749,A -85,B 0,C 180,E1 -17307.506,E2 -17307.506} C_VEL
LIN {X 0,Y 277.267,Z 540.76,A -85,B 0,C 180,E1 -17310.481,E2 -17310.481} C_VEL
LIN {X 0,Y 277.242,Z 540.76,A -85,B 0,C 180,E1 -17313.896,E2 -17313.896} C_VEL
LIN {X 0,Y 277.26,Z 540.758,A -85,B 0,C 180,E1 -17317.47,E2 -17317.47} C_VEL
LIN {X 0,Y 277.205,Z 540.766,A -85,B 0,C 180,E1 -17321.237,E2 -17321.237} C_VEL
LIN {X 0,Y 277.212,Z 540.766,A -85,B 0,C 180,E1 -17325.224,E2 -17325.224} C_VEL
LIN {X 0,Y 277.219,Z 540.764,A -85,B 0,C 180,E1 -17329.512,E2 -17329.512} C_VEL
LIN {X 0,Y 277.42,Z 540.891,A -85,B 0,C 180,E1 -17333.709,E2 -17333.709} C_VEL
LIN {X 0,Y 280.063,Z 554.585,A -85,B 0,C 180,E1 -17338.562,E2 -17338.562} C_VEL
LIN {X 0,Y 280.827,Z 558.716,A -85,B 0,C 180,E1 -17339.966,E2 -17339.966} C_VEL
LIN {X 0,Y 278.995,Z 571.89,A -85,B 0,C 180,E1 -17344.245,E2 -17344.245} C_VEL
LIN {X 0,Y 277.559,Z 584.89,A -85,B 0,C 180,E1 -17348.412,E2 -17348.412} C_VEL
LIN {X 0,Y 278.024,Z 595.266,A -85,B 0,C 180,E1 -17348.888,E2 -17348.888} C_VEL
LIN {X 0,Y 281.88,Z 652.068,A -85,B 0,C 180,E1 -17351.188,E2 -17351.188} C_VEL
LIN {X 0,Y 281.222,Z 672.799,A -85,B 0,C 180,E1 -17352.019,E2 -17352.019} C_VEL
LIN {X 0,Y 280.633,Z 684.804,A -85,B 0,C 180,E1 -17352.793,E2 -17352.793} C_VEL
LIN {X 0,Y 279.669,Z 695.765,A -85,B 0,C 180,E1 -17353.766,E2 -17353.766} C_VEL
LIN {X 0,Y 278.619,Z 706.423,A -85,B 0,C 180,E1 -17355.016,E2 -17355.016} C_VEL
LIN {X 0,Y 277.927,Z 715.024,A -85,B 0,C 180,E1 -17356.287,E2 -17356.287} C_VEL
LIN {X 0,Y 277.152,Z 723.909,A -85,B 0,C 180,E1 -17357.925,E2 -17357.925} C_VEL
LIN {X 0,Y 276.629,Z 731.847,A -85,B 0,C 180,E1 -17359.756,E2 -17359.756} C_VEL
LIN {X 0,Y 276.456,Z 738.301,A -85,B 0,C 180,E1 -17361.632,E2 -17361.632} C_VEL
LIN {X 0,Y 276.511,Z 743.232,A -85,B 0,C 180,E1 -17363.432,E2 -17363.432} C_VEL
LIN {X 0,Y 276.82,Z 747.782,A -85,B 0,C 180,E1 -17365.632,E2 -17365.632} C_VEL
LIN {X 0,Y 276.982,Z 749.988,A -85,B 0,C 180,E1 -17367.091,E2 -17367.091} C_VEL
LIN {X 0,Y 277.247,Z 751.566,A -85,B 0,C 180,E1 -17368.547,E2 -17368.547} C_VEL
LIN {X 0,Y 277.465,Z 752.589,A -85,B 0,C 180,E1 -17370,E2 -17370} C_VEL
LIN {X 0,Y 276.967,Z 752.893,A -85,B 0,C 180,E1 -17371.454,E2 -17371.454} C_VEL
LIN {X 0,Y 276.652,Z 752.72,A -85,B 0,C 180,E1 -17372.912,E2 -17372.912} C_VEL
LIN {X 0,Y 276.375,Z 751.978,A -85,B 0,C 180,E1 -17374.375,E2 -17374.375} C_VEL
LIN {X 0,Y 275.98,Z 749.76,A -85,B 0,C 180,E1 -17376.709,E2 -17376.709} C_VEL
LIN {X 0,Y 275.992,Z 746.672,A -85,B 0,C 180,E1 -17378.788,E2 -17378.788} C_VEL
LIN {X 0,Y 276.384,Z 742.138,A -85,B 0,C 180,E1 -17380.994,E2 -17380.994} C_VEL
LIN {X 0,Y 277.326,Z 736.292,A -85,B 0,C 180,E1 -17383.184,E2 -17383.184} C_VEL
LIN {X 0,Y 278.992,Z 728.823,A -85,B 0,C 180,E1 -17385.337,E2 -17385.337} C_VEL
LIN {X 0,Y 280.664,Z 721.102,A -85,B 0,C 180,E1 -17387.111,E2 -17387.111} C_VEL
LIN {X 0,Y 282.892,Z 711.573,A -85,B 0,C 180,E1 -17388.842,E2 -17388.842} C_VEL
LIN {X 0,Y 285.225,Z 701.094,A -85,B 0,C 180,E1 -17390.355,E2 -17390.355} C_VEL
LIN {X 0,Y 287.476,Z 689.635,A -85,B 0,C 180,E1 -17391.645,E2 -17391.645} C_VEL
LIN {X 0,Y 289.611,Z 676.695,A -85,B 0,C 180,E1 -17392.736,E2 -17392.736} C_VEL
LIN {X 0,Y 291.281,Z 663.612,A -85,B 0,C 180,E1 -17393.519,E2 -17393.519} C_VEL
LIN {X 0,Y 291.935,Z 652.581,A -85,B 0,C 180,E1 -17394.014,E2 -17394.014} C_VEL
LIN {X 0,Y 291.456,Z 629.456,A -85,B 0,C 180,E1 -17395.06,E2 -17395.06} C_VEL
LIN {X 0,Y 290.163,Z 613.939,A -85,B 0,C 180,E1 -17395.943,E2 -17395.943} C_VEL
LIN {X 0,Y 287.919,Z 597.206,A -85,B 0,C 180,E1 -17397.058,E2 -17397.058} C_VEL
LIN {X 0,Y 285.101,Z 581.952,A -85,B 0,C 180,E1 -17398.277,E2 -17398.277} C_VEL
LIN {X 0,Y 282.068,Z 568.241,A -85,B 0,C 180,E1 -17399.527,E2 -17399.527} C_VEL
LIN {X 0,Y 281.152,Z 563.453,A -85,B 0,C 180,E1 -17400.047,E2 -17400.047} C_VEL
LIN {X 0,Y 281.17,Z 559.954,A -85,B 0,C 180,E1 -17401.241,E2 -17401.241} C_VEL
LIN {X 0,Y 279.713,Z 551.602,A -85,B 0,C 180,E1 -17404.584,E2 -17404.584} C_VEL
LIN {X 0,Y 277.83,Z 543.14,A -85,B 0,C 180,E1 -17408.356,E2 -17408.356} C_VEL
LIN {X 0,Y 277.286,Z 540.82,A -85,B 0,C 180,E1 -17409.536,E2 -17409.536} C_VEL
LIN {X 0,Y 277.231,Z 540.765,A -85,B 0,C 180,E1 -17413.192,E2 -17413.192} C_VEL
LIN {X 0,Y 277.267,Z 540.753,A -85,B 0,C 180,E1 -17417.312,E2 -17417.312} C_VEL
LIN {X 0,Y 277.263,Z 540.753,A -85,B 0,C 180,E1 -17420.677,E2 -17420.677} C_VEL
LIN {X 0,Y 277.3,Z 540.747,A -85,B 0,C 180,E1 -17424.344,E2 -17424.344} C_VEL
LIN {X 0,Y 277.24,Z 540.756,A -85,B 0,C 180,E1 -17427.836,E2 -17427.836} C_VEL
LIN {X 0,Y 277.266,Z 540.754,A -85,B 0,C 180,E1 -17431.21,E2 -17431.21} C_VEL
LIN {X 0,Y 277.307,Z 540.75,A -85,B 0,C 180,E1 -17434.479,E2 -17434.479} C_VEL
LIN {X 0,Y 277.284,Z 540.755,A -85,B 0,C 180,E1 -17437.655,E2 -17437.655} C_VEL
LIN {X 0,Y 277.338,Z 540.751,A -85,B 0,C 180,E1 -17440.766,E2 -17440.766} C_VEL
LIN {X 0,Y 277.422,Z 540.738,A -85,B 0,C 180,E1 -17445.326,E2 -17445.326} C_VEL
LIN {X 0,Y 277.5,Z 540.94,A -85,B 0,C 180,E1 -17449.153,E2 -17449.153} C_VEL
LIN {X 0,Y 277.692,Z 541.837,A -85,B 0,C 180,E1 -17449.465,E2 -17449.465} C_VEL
LIN {X 0,Y 279.197,Z 544.508,A -85,B 0,C 180,E1 -17449.95,E2 -17449.95} C_VEL
LIN {X 0,Y 280.739,Z 546.101,A -85,B 0,C 180,E1 -17450.369,E2 -17450.369} C_VEL
LIN {X 0,Y 282.953,Z 549.556,A -85,B 0,C 180,E1 -17450.979,E2 -17450.979} C_VEL
LIN {X 0,Y 287.735,Z 557.068,A -85,B 0,C 180,E1 -17452.242,E2 -17452.242} C_VEL
LIN {X 0,Y 295.458,Z 571.072,A -85,B 0,C 180,E1 -17454.113,E2 -17454.113} C_VEL
LIN {X 0,Y 296.593,Z 573.405,A -85,B 0,C 180,E1 -17454.381,E2 -17454.381} C_VEL
LIN {X 0,Y 296.403,Z 589.987,A -85,B 0,C 180,E1 -17455.061,E2 -17455.061} C_VEL
LIN {X 0,Y 295.814,Z 601.581,A -85,B 0,C 180,E1 -17455.79,E2 -17455.79} C_VEL
LIN {X 0,Y 294.801,Z 612.945,A -85,B 0,C 180,E1 -17456.755,E2 -17456.755} C_VEL
LIN {X 0,Y 293.388,Z 623.789,A -85,B 0,C 180,E1 -17457.941,E2 -17457.941} C_VEL
LIN {X 0,Y 291.554,Z 634.68,A -85,B 0,C 180,E1 -17459.483,E2 -17459.483} C_VEL
LIN {X 0,Y 289.807,Z 643.484,A -85,B 0,C 180,E1 -17461.043,E2 -17461.043} C_VEL
LIN {X 0,Y 287.883,Z 651.494,A -85,B 0,C 180,E1 -17462.799,E2 -17462.799} C_VEL
LIN {X 0,Y 285.801,Z 659.206,A -85,B 0,C 180,E1 -17464.938,E2 -17464.938} C_VEL
LIN {X 0,Y 283.923,Z 665.222,A -85,B 0,C 180,E1 -17467.11,E2 -17467.11} C_VEL
LIN {X 0,Y 282.279,Z 669.845,A -85,B 0,C 180,E1 -17469.314,E2 -17469.314} C_VEL
LIN {X 0,Y 280.89,Z 673.249,A -85,B 0,C 180,E1 -17471.547,E2 -17471.547} C_VEL
LIN {X 0,Y 280.101,Z 674.887,A -85,B 0,C 180,E1 -17473.052,E2 -17473.052} C_VEL
LIN {X 0,Y 279.411,Z 676.01,A -85,B 0,C 180,E1 -17474.569,E2 -17474.569} C_VEL
LIN {X 0,Y 278.671,Z 676.771,A -85,B 0,C 180,E1 -17476.6,E2 -17476.6} C_VEL
LIN {X 0,Y 278.019,Z 676.52,A -85,B 0,C 180,E1 -17479.186,E2 -17479.186} C_VEL
LIN {X 0,Y 277.768,Z 675.685,A -85,B 0,C 180,E1 -17480.746,E2 -17480.746} C_VEL
LIN {X 0,Y 277.622,Z 674.372,A -85,B 0,C 180,E1 -17482.317,E2 -17482.317} C_VEL
LIN {X 0,Y 277.603,Z 671.951,A -85,B 0,C 180,E1 -17484.304,E2 -17484.304} C_VEL
LIN {X 0,Y 277.813,Z 668.682,A -85,B 0,C 180,E1 -17486.277,E2 -17486.277} C_VEL
LIN {X 0,Y 278.171,Z 663.442,A -85,B 0,C 180,E1 -17488.688,E2 -17488.688} C_VEL
LIN {X 0,Y 278.743,Z 656.863,A -85,B 0,C 180,E1 -17490.994,E2 -17490.994} C_VEL
LIN {X 0,Y 279.504,Z 649.108,A -85,B 0,C 180,E1 -17493.155,E2 -17493.155} C_VEL
LIN {X 0,Y 280.397,Z 639.875,A -85,B 0,C 180,E1 -17495.204,E2 -17495.204} C_VEL
LIN {X 0,Y 281.256,Z 630.384,A -85,B 0,C 180,E1 -17496.909,E2 -17496.909} C_VEL
LIN {X 0,Y 282.158,Z 619.238,A -85,B 0,C 180,E1 -17498.514,E2 -17498.514} C_VEL
LIN {X 0,Y 282.878,Z 607.956,A -85,B 0,C 180,E1 -17499.801,E2 -17499.801} C_VEL
LIN {X 0,Y 283.535,Z 596.352,A -85,B 0,C 180,E1 -17500.826,E2 -17500.826} C_VEL
LIN {X 0,Y 283.974,Z 582.764,A -85,B 0,C 180,E1 -17501.692,E2 -17501.692} C_VEL
LIN {X 0,Y 284.076,Z 569.557,A -85,B 0,C 180,E1 -17502.241,E2 -17502.241} C_VEL
LIN {X 0,Y 283.916,Z 561.637,A -85,B 0,C 180,E1 -17502.508,E2 -17502.508} C_VEL
LIN {X 0,Y 277.489,Z 541.729,A -85,B 0,C 180,E1 -17503.51,E2 -17503.51} C_VEL
LIN {X 0,Y 277.303,Z 540.83,A -85,B 0,C 180,E1 -17503.805,E2 -17503.805} C_VEL
LIN {X 0,Y 277.27,Z 540.762,A -85,B 0,C 180,E1 -17507.314,E2 -17507.314} C_VEL
LIN {X 0,Y 277.268,Z 540.758,A -85,B 0,C 180,E1 -17510.679,E2 -17510.679} C_VEL
LIN {X 0,Y 277.306,Z 540.753,A -85,B 0,C 180,E1 -17514.346,E2 -17514.346} C_VEL
LIN {X 0,Y 277.246,Z 540.762,A -85,B 0,C 180,E1 -17517.838,E2 -17517.838} C_VEL
LIN {X 0,Y 277.291,Z 540.757,A -85,B 0,C 180,E1 -17521.214,E2 -17521.214} C_VEL
LIN {X 0,Y 277.316,Z 540.751,A -85,B 0,C 180,E1 -17524.481,E2 -17524.481} C_VEL
LIN {X 0,Y 277.285,Z 540.759,A -85,B 0,C 180,E1 -17527.655,E2 -17527.655} C_VEL
LIN {X 0,Y 277.331,Z 540.749,A -85,B 0,C 180,E1 -17530.766,E2 -17530.766} C_VEL
LIN {X 0,Y 277.418,Z 540.74,A -85,B 0,C 180,E1 -17535.325,E2 -17535.325} C_VEL
LIN {X 0,Y 277.464,Z 540.736,A -85,B 0,C 180,E1 -17539.787,E2 -17539.787} C_VEL
LIN {X 0,Y 277.615,Z 540.712,A -85,B 0,C 180,E1 -17542.728,E2 -17542.728} C_VEL
LIN {X 0,Y 277.825,Z 540.687,A -85,B 0,C 180,E1 -17548.551,E2 -17548.551} C_VEL
LIN {X 0,Y 277.825,Z 540.689,A -85,B 0,C 180,E1 -17551.45,E2 -17551.45} C_VEL
LIN {X 0,Y 277.615,Z 540.715,A -85,B 0,C 180,E1 -17557.272,E2 -17557.272} C_VEL
LIN {X 0,Y 277.461,Z 540.733,A -85,B 0,C 180,E1 -17560.213,E2 -17560.213} C_VEL
LIN {X 0,Y 277.439,Z 540.736,A -85,B 0,C 180,E1 -17564.674,E2 -17564.674} C_VEL
LIN {X 0,Y 277.348,Z 540.746,A -85,B 0,C 180,E1 -17569.233,E2 -17569.233} C_VEL
LIN {X 0,Y 277.295,Z 540.757,A -85,B 0,C 180,E1 -17574.157,E2 -17574.157} C_VEL
LIN {X 0,Y 277.326,Z 540.75,A -85,B 0,C 180,E1 -17577.504,E2 -17577.504} C_VEL
LIN {X 0,Y 277.274,Z 540.757,A -85,B 0,C 180,E1 -17580.48,E2 -17580.48} C_VEL
LIN {X 0,Y 277.256,Z 540.763,A -85,B 0,C 180,E1 -17583.894,E2 -17583.894} C_VEL
LIN {X 0,Y 277.291,Z 540.753,A -85,B 0,C 180,E1 -17587.465,E2 -17587.465} C_VEL
LIN {X 0,Y 277.266,Z 540.757,A -85,B 0,C 180,E1 -17591.225,E2 -17591.225} C_VEL
LIN {X 0,Y 277.243,Z 540.759,A -85,B 0,C 180,E1 -17595.217,E2 -17595.217} C_VEL
LIN {X 0,Y 277.224,Z 540.763,A -85,B 0,C 180,E1 -17599.51,E2 -17599.51} C_VEL
LIN {X 0,Y 277.272,Z 540.758,A -85,B 0,C 180,E1 -17602.531,E2 -17602.531} C_VEL
LIN {X 0,Y 277.245,Z 540.763,A -85,B 0,C 180,E1 -17606.103,E2 -17606.103} C_VEL
LIN {X 0,Y 277.259,Z 540.759,A -85,B 0,C 180,E1 -17609.538,E2 -17609.538} C_VEL
LIN {X 0,Y 277.356,Z 540.745,A -85,B 0,C 180,E1 -17612.863,E2 -17612.863} C_VEL
LIN {X 0,Y 277.325,Z 540.752,A -85,B 0,C 180,E1 -17616.079,E2 -17616.079} C_VEL
LIN {X 0,Y 277.342,Z 540.748,A -85,B 0,C 180,E1 -17620.765,E2 -17620.765} C_VEL
LIN {X 0,Y 277.424,Z 540.737,A -85,B 0,C 180,E1 -17625.325,E2 -17625.325} C_VEL
LIN {X 0,Y 277.502,Z 540.728,A -85,B 0,C 180,E1 -17629.788,E2 -17629.788} C_VEL
LIN {X 0,Y 277.648,Z 540.712,A -85,B 0,C 180,E1 -17632.728,E2 -17632.728} C_VEL
LIN {X 0,Y 277.816,Z 540.692,A -85,B 0,C 180,E1 -17638.55,E2 -17638.55} C_VEL
LIN {X 0,Y 277.8,Z 540.689,A -85,B 0,C 180,E1 -17641.561,E2 -17641.561} C_VEL
LIN {X 0,Y 277.643,Z 540.71,A -85,B 0,C 180,E1 -17647.271,E2 -17647.271} C_VEL
LIN {X 0,Y 277.607,Z 540.713,A -85,B 0,C 180,E1 -17647.872,E2 -17647.872} C_VEL
LIN {X 0,Y 276.892,Z 540.805,A -85,B 0,C 180,E1 -17649.082,E2 -17649.082} C_VEL
LIN {X 0,Y 273.937,Z 541.173,A -85,B 0,C 180,E1 -17651.051,E2 -17651.051} C_VEL
LIN {X 0,Y 271.46,Z 541.485,A -85,B 0,C 180,E1 -17652.651,E2 -17652.651} C_VEL
LIN {X 0,Y 270.42,Z 541.611,A -85,B 0,C 180,E1 -17653.894,E2 -17653.894} C_VEL
LIN {X 0,Y 270.347,Z 541.617,A -85,B 0,C 180,E1 -17654.315,E2 -17654.315} C_VEL
LIN {X 0,Y 270.282,Z 541.627,A -85,B 0,C 180,E1 -17658.181,E2 -17658.181} C_VEL
LIN {X 0,Y 270.208,Z 541.637,A -85,B 0,C 180,E1 -17661.354,E2 -17661.354} C_VEL
LIN {X 0,Y 270.233,Z 541.637,A -85,B 0,C 180,E1 -17664.589,E2 -17664.589} C_VEL
LIN {X 0,Y 270.267,Z 541.628,A -85,B 0,C 180,E1 -17667.909,E2 -17667.909} C_VEL
LIN {X 0,Y 270.179,Z 541.641,A -85,B 0,C 180,E1 -17671.348,E2 -17671.348} C_VEL
LIN {X 0,Y 270.196,Z 541.64,A -85,B 0,C 180,E1 -17674.906,E2 -17674.906} C_VEL
LIN {X 0,Y 270.193,Z 541.642,A -85,B 0,C 180,E1 -17678.711,E2 -17678.711} C_VEL
LIN {X 0,Y 270.167,Z 541.643,A -85,B 0,C 180,E1 -17683.251,E2 -17683.251} C_VEL
LIN {X 0,Y 270.171,Z 541.642,A -85,B 0,C 180,E1 -17687.443,E2 -17687.443} C_VEL
LIN {X 0,Y 270.204,Z 541.639,A -85,B 0,C 180,E1 -17691.375,E2 -17691.375} C_VEL
LIN {X 0,Y 270.366,Z 541.713,A -85,B 0,C 180,E1 -17693.546,E2 -17693.546} C_VEL
LIN {X 0,Y 272.788,Z 554.484,A -85,B 0,C 180,E1 -17698.233,E2 -17698.233} C_VEL
LIN {X 0,Y 273.728,Z 559.419,A -85,B 0,C 180,E1 -17699.957,E2 -17699.957} C_VEL
LIN {X 0,Y 272.006,Z 571.332,A -85,B 0,C 180,E1 -17703.945,E2 -17703.945} C_VEL
LIN {X 0,Y 270.583,Z 583.682,A -85,B 0,C 180,E1 -17708.027,E2 -17708.027} C_VEL
LIN {X 0,Y 270.879,Z 591.252,A -85,B 0,C 180,E1 -17708.402,E2 -17708.402} C_VEL
LIN {X 0,Y 274.859,Z 653.675,A -85,B 0,C 180,E1 -17711.007,E2 -17711.007} C_VEL
LIN {X 0,Y 274.229,Z 672.321,A -85,B 0,C 180,E1 -17711.79,E2 -17711.79} C_VEL
LIN {X 0,Y 273.499,Z 685.768,A -85,B 0,C 180,E1 -17712.716,E2 -17712.716} C_VEL
LIN {X 0,Y 272.372,Z 697.838,A -85,B 0,C 180,E1 -17713.896,E2 -17713.896} C_VEL
LIN {X 0,Y 271.438,Z 707.827,A -85,B 0,C 180,E1 -17715.186,E2 -17715.186} C_VEL
LIN {X 0,Y 270.654,Z 717.033,A -85,B 0,C 180,E1 -17716.676,E2 -17716.676} C_VEL
LIN {X 0,Y 269.901,Z 725.303,A -85,B 0,C 180,E1 -17718.358,E2 -17718.358} C_VEL
LIN {X 0,Y 269.491,Z 732.771,A -85,B 0,C 180,E1 -17720.241,E2 -17720.241} C_VEL
LIN {X 0,Y 269.411,Z 739.533,A -85,B 0,C 180,E1 -17722.429,E2 -17722.429} C_VEL
LIN {X 0,Y 269.695,Z 744.977,A -85,B 0,C 180,E1 -17724.767,E2 -17724.767} C_VEL
LIN {X 0,Y 269.964,Z 748.63,A -85,B 0,C 180,E1 -17727.015,E2 -17727.015} C_VEL
LIN {X 0,Y 270.224,Z 750.303,A -85,B 0,C 180,E1 -17728.51,E2 -17728.51} C_VEL
LIN {X 0,Y 270.474,Z 751.386,A -85,B 0,C 180,E1 -17730,E2 -17730} C_VEL
LIN {X 0,Y 269.961,Z 751.774,A -85,B 0,C 180,E1 -17731.492,E2 -17731.492} C_VEL
LIN {X 0,Y 269.594,Z 751.651,A -85,B 0,C 180,E1 -17732.988,E2 -17732.988} C_VEL
LIN {X 0,Y 269.303,Z 751.003,A -85,B 0,C 180,E1 -17734.49,E2 -17734.49} C_VEL
LIN {X 0,Y 268.907,Z 749.072,A -85,B 0,C 180,E1 -17736.715,E2 -17736.715} C_VEL
LIN {X 0,Y 268.949,Z 745.92,A -85,B 0,C 180,E1 -17739.02,E2 -17739.02} C_VEL
LIN {X 0,Y 269.369,Z 741.588,A -85,B 0,C 180,E1 -17741.284,E2 -17741.284} C_VEL
LIN {X 0,Y 270.409,Z 735.881,A -85,B 0,C 180,E1 -17743.527,E2 -17743.527} C_VEL
LIN {X 0,Y 272.156,Z 728.637,A -85,B 0,C 180,E1 -17745.732,E2 -17745.732} C_VEL
LIN {X 0,Y 274.308,Z 719.5,A -85,B 0,C 180,E1 -17747.905,E2 -17747.905} C_VEL
LIN {X 0,Y 276.748,Z 709.961,A -85,B 0,C 180,E1 -17749.662,E2 -17749.662} C_VEL
LIN {X 0,Y 279.272,Z 699.066,A -85,B 0,C 180,E1 -17751.242,E2 -17751.242} C_VEL
LIN {X 0,Y 281.591,Z 687.795,A -85,B 0,C 180,E1 -17752.512,E2 -17752.512} C_VEL
LIN {X 0,Y 283.87,Z 674.553,A -85,B 0,C 180,E1 -17753.625,E2 -17753.625} C_VEL
LIN {X 0,Y 285.7,Z 660.371,A -85,B 0,C 180,E1 -17754.472,E2 -17754.472} C_VEL
LIN {X 0,Y 286.146,Z 649.899,A -85,B 0,C 180,E1 -17754.961,E2 -17754.961} C_VEL
LIN {X 0,Y 285.764,Z 630.188,A -85,B 0,C 180,E1 -17755.9,E2 -17755.9} C_VEL
LIN {X 0,Y 284.607,Z 615.846,A -85,B 0,C 180,E1 -17756.743,E2 -17756.743} C_VEL
LIN {X 0,Y 282.728,Z 600.496,A -85,B 0,C 180,E1 -17757.803,E2 -17757.803} C_VEL
LIN {X 0,Y 279.934,Z 584.371,A -85,B 0,C 180,E1 -17759.13,E2 -17759.13} C_VEL
LIN {X 0,Y 277.169,Z 571.344,A -85,B 0,C 180,E1 -17760.371,E2 -17760.371} C_VEL
LIN {X 0,Y 275.776,Z 565.805,A -85,B 0,C 180,E1 -17760.975,E2 -17760.975} C_VEL
LIN {X 0,Y 274.188,Z 560.822,A -85,B 0,C 180,E1 -17761.709,E2 -17761.709} C_VEL
LIN {X 0,Y 272.937,Z 553.805,A -85,B 0,C 180,E1 -17764.515,E2 -17764.515} C_VEL
LIN {X 0,Y 271.293,Z 546.184,A -85,B 0,C 180,E1 -17767.977,E2 -17767.977} C_VEL
LIN {X 0,Y 270.206,Z 541.66,A -85,B 0,C 180,E1 -17770.328,E2 -17770.328} C_VEL
LIN {X 0,Y 270.184,Z 541.636,A -85,B 0,C 180,E1 -17774.612,E2 -17774.612} C_VEL
LIN {X 0,Y 270.262,Z 541.63,A -85,B 0,C 180,E1 -17778.947,E2 -17778.947} C_VEL
LIN {X 0,Y 270.239,Z 541.632,A -85,B 0,C 180,E1 -17783.263,E2 -17783.263} C_VEL
LIN {X 0,Y 270.199,Z 541.633,A -85,B 0,C 180,E1 -17786.893,E2 -17786.893} C_VEL
LIN {X 0,Y 270.191,Z 541.634,A -85,B 0,C 180,E1 -17790.383,E2 -17790.383} C_VEL
LIN {X 0,Y 270.257,Z 541.625,A -85,B 0,C 180,E1 -17793.764,E2 -17793.764} C_VEL
LIN {X 0,Y 270.229,Z 541.63,A -85,B 0,C 180,E1 -17797.039,E2 -17797.039} C_VEL
LIN {X 0,Y 270.296,Z 541.624,A -85,B 0,C 180,E1 -17800.245,E2 -17800.245} C_VEL
LIN {X 0,Y 270.39,Z 541.612,A -85,B 0,C 180,E1 -17804.935,E2 -17804.935} C_VEL
LIN {X 0,Y 270.386,Z 541.867,A -85,B 0,C 180,E1 -17807.475,E2 -17807.475} C_VEL
LIN {X 0,Y 270.66,Z 542.936,A -85,B 0,C 180,E1 -17807.821,E2 -17807.821} C_VEL
LIN {X 0,Y 272.168,Z 545.481,A -85,B 0,C 180,E1 -17808.369,E2 -17808.369} C_VEL
LIN {X 0,Y 273.904,Z 547.218,A -85,B 0,C 180,E1 -17808.877,E2 -17808.877} C_VEL
LIN {X 0,Y 275.613,Z 550.068,A -85,B 0,C 180,E1 -17809.424,E2 -17809.424} C_VEL
LIN {X 0,Y 277.088,Z 551.853,A -85,B 0,C 180,E1 -17809.852,E2 -17809.852} C_VEL
LIN {X 0,Y 282.312,Z 559.932,A -85,B 0,C 180,E1 -17811.32,E2 -17811.32} C_VEL
LIN {X 0,Y 290.383,Z 574.584,A -85,B 0,C 180,E1 -17813.417,E2 -17813.417} C_VEL
LIN {X 0,Y 291.17,Z 576.302,A -85,B 0,C 180,E1 -17813.617,E2 -17813.617} C_VEL
LIN {X 0,Y 290.756,Z 591.857,A -85,B 0,C 180,E1 -17814.274,E2 -17814.274} C_VEL
LIN {X 0,Y 289.981,Z 604.765,A -85,B 0,C 180,E1 -17815.144,E2 -17815.144} C_VEL
LIN {X 0,Y 288.776,Z 616.406,A -85,B 0,C 180,E1 -17816.198,E2 -17816.198} C_VEL
LIN {X 0,Y 287.101,Z 627.793,A -85,B 0,C 180,E1 -17817.545,E2 -17817.545} C_VEL
LIN {X 0,Y 285.159,Z 638.159,A -85,B 0,C 180,E1 -17819.118,E2 -17819.118} C_VEL
LIN {X 0,Y 283.308,Z 646.504,A -85,B 0,C 180,E1 -17820.711,E2 -17820.711} C_VEL
LIN {X 0,Y 281.367,Z 653.883,A -85,B 0,C 180,E1 -17822.436,E2 -17822.436} C_VEL
LIN {X 0,Y 279.434,Z 660.429,A -85,B 0,C 180,E1 -17824.328,E2 -17824.328} C_VEL
LIN {X 0,Y 277.429,Z 666.446,A -85,B 0,C 180,E1 -17826.546,E2 -17826.546} C_VEL
LIN {X 0,Y 275.682,Z 671.057,A -85,B 0,C 180,E1 -17828.799,E2 -17828.799} C_VEL
LIN {X 0,Y 274.68,Z 673.455,A -85,B 0,C 180,E1 -17830.318,E2 -17830.318} C_VEL
LIN {X 0,Y 273.438,Z 675.863,A -85,B 0,C 180,E1 -17832.402,E2 -17832.402} C_VEL
LIN {X 0,Y 272.244,Z 677.535,A -85,B 0,C 180,E1 -17834.961,E2 -17834.961} C_VEL
LIN {X 0,Y 271.606,Z 677.967,A -85,B 0,C 180,E1 -17836.789,E2 -17836.789} C_VEL
LIN {X 0,Y 271.235,Z 677.847,A -85,B 0,C 180,E1 -17838.116,E2 -17838.116} C_VEL
LIN {X 0,Y 270.715,Z 676.538,A -85,B 0,C 180,E1 -17840.842,E2 -17840.842} C_VEL
LIN {X 0,Y 270.56,Z 673.562,A -85,B 0,C 180,E1 -17843.743,E2 -17843.743} C_VEL
LIN {X 0,Y 270.764,Z 669.694,A -85,B 0,C 180,E1 -17846.185,E2 -17846.185} C_VEL
LIN {X 0,Y 271.111,Z 664.192,A -85,B 0,C 180,E1 -17848.751,E2 -17848.751} C_VEL
LIN {X 0,Y 271.707,Z 657.404,A -85,B 0,C 180,E1 -17851.154,E2 -17851.154} C_VEL
LIN {X 0,Y 272.452,Z 650.036,A -85,B 0,C 180,E1 -17853.241,E2 -17853.241} C_VEL
LIN {X 0,Y 273.369,Z 640.774,A -85,B 0,C 180,E1 -17855.341,E2 -17855.341} C_VEL
LIN {X 0,Y 274.187,Z 631.796,A -85,B 0,C 180,E1 -17856.999,E2 -17856.999} C_VEL
LIN {X 0,Y 275.066,Z 621.715,A -85,B 0,C 180,E1 -17858.521,E2 -17858.521} C_VEL
LIN {X 0,Y 275.825,Z 610.204,A -85,B 0,C 180,E1 -17859.899,E2 -17859.899} C_VEL
LIN {X 0,Y 276.526,Z 598.213,A -85,B 0,C 180,E1 -17861.011,E2 -17861.011} C_VEL
LIN {X 0,Y 276.958,Z 585.009,A -85,B 0,C 180,E1 -17861.898,E2 -17861.898} C_VEL
LIN {X 0,Y 277.166,Z 571.774,A -85,B 0,C 180,E1 -17862.483,E2 -17862.483} C_VEL
LIN {X 0,Y 276.972,Z 563.058,A -85,B 0,C 180,E1 -17862.787,E2 -17862.787} C_VEL
LIN {X 0,Y 270.4,Z 542.463,A -85,B 0,C 180,E1 -17863.86,E2 -17863.86} C_VEL
LIN {X 0,Y 270.22,Z 541.699,A -85,B 0,C 180,E1 -17864.156,E2 -17864.156} C_VEL
LIN {X 0,Y 270.222,Z 541.64,A -85,B 0,C 180,E1 -17867.453,E2 -17867.453} C_VEL
LIN {X 0,Y 270.245,Z 541.637,A -85,B 0,C 180,E1 -17871.382,E2 -17871.382} C_VEL
LIN {X 0,Y 270.217,Z 541.638,A -85,B 0,C 180,E1 -17875.098,E2 -17875.098} C_VEL
LIN {X 0,Y 270.202,Z 541.64,A -85,B 0,C 180,E1 -17879.132,E2 -17879.132} C_VEL
LIN {X 0,Y 270.267,Z 541.63,A -85,B 0,C 180,E1 -17882.147,E2 -17882.147} C_VEL
LIN {X 0,Y 270.28,Z 541.632,A -85,B 0,C 180,E1 -17885.52,E2 -17885.52} C_VEL
LIN {X 0,Y 270.277,Z 541.628,A -85,B 0,C 180,E1 -17890.243,E2 -17890.243} C_VEL
LIN {X 0,Y 270.377,Z 541.615,A -85,B 0,C 180,E1 -17894.934,E2 -17894.934} C_VEL
LIN {X 0,Y 270.416,Z 541.614,A -85,B 0,C 180,E1 -17899.518,E2 -17899.518} C_VEL
LIN {X 0,Y 270.575,Z 541.589,A -85,B 0,C 180,E1 -17902.538,E2 -17902.538} C_VEL
LIN {X 0,Y 270.79,Z 541.564,A -85,B 0,C 180,E1 -17908.513,E2 -17908.513} C_VEL
LIN {X 0,Y 270.791,Z 541.565,A -85,B 0,C 180,E1 -17911.487,E2 -17911.487} C_VEL
LIN {X 0,Y 270.575,Z 541.593,A -85,B 0,C 180,E1 -17917.462,E2 -17917.462} C_VEL
LIN {X 0,Y 270.414,Z 541.61,A -85,B 0,C 180,E1 -17920.482,E2 -17920.482} C_VEL
LIN {X 0,Y 270.407,Z 541.612,A -85,B 0,C 180,E1 -17925.064,E2 -17925.064} C_VEL
LIN {X 0,Y 270.304,Z 541.626,A -85,B 0,C 180,E1 -17929.755,E2 -17929.755} C_VEL
LIN {X 0,Y 270.241,Z 541.633,A -85,B 0,C 180,E1 -17934.588,E2 -17934.588} C_VEL
LIN {X 0,Y 270.272,Z 541.631,A -85,B 0,C 180,E1 -17937.908,E2 -17937.908} C_VEL
LIN {X 0,Y 270.186,Z 541.64,A -85,B 0,C 180,E1 -17941.347,E2 -17941.347} C_VEL
LIN {X 0,Y 270.217,Z 541.635,A -85,B 0,C 180,E1 -17944.902,E2 -17944.902} C_VEL
LIN {X 0,Y 270.223,Z 541.635,A -85,B 0,C 180,E1 -17948.716,E2 -17948.716} C_VEL
LIN {X 0,Y 270.223,Z 541.636,A -85,B 0,C 180,E1 -17952.547,E2 -17952.547} C_VEL
LIN {X 0,Y 270.189,Z 541.639,A -85,B 0,C 180,E1 -17956.745,E2 -17956.745} C_VEL
LIN {X 0,Y 270.206,Z 541.637,A -85,B 0,C 180,E1 -17961.373,E2 -17961.373} C_VEL
LIN {X 0,Y 270.201,Z 541.636,A -85,B 0,C 180,E1 -17965.094,E2 -17965.094} C_VEL
LIN {X 0,Y 270.198,Z 541.638,A -85,B 0,C 180,E1 -17969.129,E2 -17969.129} C_VEL
LIN {X 0,Y 270.261,Z 541.633,A -85,B 0,C 180,E1 -17972.145,E2 -17972.145} C_VEL
LIN {X 0,Y 270.274,Z 541.628,A -85,B 0,C 180,E1 -17975.518,E2 -17975.518} C_VEL
LIN {X 0,Y 270.299,Z 541.629,A -85,B 0,C 180,E1 -17980.244,E2 -17980.244} C_VEL
LIN {X 0,Y 270.392,Z 541.614,A -85,B 0,C 180,E1 -17984.934,E2 -17984.934} C_VEL
LIN {X 0,Y 270.437,Z 541.607,A -85,B 0,C 180,E1 -17989.518,E2 -17989.518} C_VEL
LIN {X 0,Y 270.606,Z 541.59,A -85,B 0,C 180,E1 -17992.538,E2 -17992.538} C_VEL
LIN {X 0,Y 270.782,Z 541.568,A -85,B 0,C 180,E1 -17998.512,E2 -17998.512} C_VEL
LIN {X 0,Y 270.781,Z 541.564,A -85,B 0,C 180,E1 -18001.487,E2 -18001.487} C_VEL
LIN {X 0,Y 270.602,Z 541.587,A -85,B 0,C 180,E1 -18007.461,E2 -18007.461} C_VEL
LIN {X 0,Y 270.436,Z 541.611,A -85,B 0,C 180,E1 -18010.481,E2 -18010.481} C_VEL
LIN {X 0,Y 270.347,Z 541.617,A -85,B 0,C 180,E1 -18014.315,E2 -18014.315} C_VEL
LIN {X 0,Y 269.718,Z 541.699,A -85,B 0,C 180,E1 -18015.559,E2 -18015.559} C_VEL
LIN {X 0,Y 266.892,Z 542.058,A -85,B 0,C 180,E1 -18017.585,E2 -18017.585} C_VEL
LIN {X 0,Y 264.433,Z 542.366,A -85,B 0,C 180,E1 -18019.231,E2 -18019.231} C_VEL
LIN {X 0,Y 263.319,Z 542.5,A -85,B 0,C 180,E1 -18020.508,E2 -18020.508} C_VEL
LIN {X 0,Y 263.199,Z 542.512,A -85,B 0,C 180,E1 -18020.941,E2 -18020.941} C_VEL
LIN {X 0,Y 263.188,Z 542.511,A -85,B 0,C 180,E1 -18025.293,E2 -18025.293} C_VEL
LIN {X 0,Y 263.175,Z 542.516,A -85,B 0,C 180,E1 -18028.73,E2 -18028.73} C_VEL
LIN {X 0,Y 263.128,Z 542.52,A -85,B 0,C 180,E1 -18032.288,E2 -18032.288} C_VEL
LIN {X 0,Y 263.177,Z 542.515,A -85,B 0,C 180,E1 -18036.763,E2 -18036.763} C_VEL
LIN {X 0,Y 263.121,Z 542.519,A -85,B 0,C 180,E1 -18041.594,E2 -18041.594} C_VEL
LIN {X 0,Y 263.124,Z 542.519,A -85,B 0,C 180,E1 -18046.017,E2 -18046.017} C_VEL
LIN {X 0,Y 263.112,Z 542.521,A -85,B 0,C 180,E1 -18050.13,E2 -18050.13} C_VEL
LIN {X 0,Y 263.335,Z 542.653,A -85,B 0,C 180,E1 -18053.491,E2 -18053.491} C_VEL
LIN {X 0,Y 265.645,Z 554.804,A -85,B 0,C 180,E1 -18058.054,E2 -18058.054} C_VEL
LIN {X 0,Y 266.636,Z 560.059,A -85,B 0,C 180,E1 -18059.948,E2 -18059.948} C_VEL
LIN {X 0,Y 264.664,Z 573.338,A -85,B 0,C 180,E1 -18064.534,E2 -18064.534} C_VEL
LIN {X 0,Y 263.611,Z 582.451,A -85,B 0,C 180,E1 -18067.621,E2 -18067.621} C_VEL
LIN {X 0,Y 263.779,Z 588.551,A -85,B 0,C 180,E1 -18067.945,E2 -18067.945} C_VEL
LIN {X 0,Y 267.854,Z 654.274,A -85,B 0,C 180,E1 -18070.78,E2 -18070.78} C_VEL
LIN {X 0,Y 267.303,Z 670.957,A -85,B 0,C 180,E1 -18071.51,E2 -18071.51} C_VEL
LIN {X 0,Y 266.623,Z 683.167,A -85,B 0,C 180,E1 -18072.354,E2 -18072.354} C_VEL
LIN {X 0,Y 265.774,Z 693.123,A -85,B 0,C 180,E1 -18073.288,E2 -18073.288} C_VEL
LIN {X 0,Y 264.537,Z 705.201,A -85,B 0,C 180,E1 -18074.791,E2 -18074.791} C_VEL
LIN {X 0,Y 263.75,Z 714.659,A -85,B 0,C 180,E1 -18076.321,E2 -18076.321} C_VEL
LIN {X 0,Y 262.995,Z 723.226,A -85,B 0,C 180,E1 -18078.048,E2 -18078.048} C_VEL
LIN {X 0,Y 262.531,Z 730.844,A -85,B 0,C 180,E1 -18079.979,E2 -18079.979} C_VEL
LIN {X 0,Y 262.397,Z 736.977,A -85,B 0,C 180,E1 -18081.917,E2 -18081.917} C_VEL
LIN {X 0,Y 262.531,Z 741.815,A -85,B 0,C 180,E1 -18083.853,E2 -18083.853} C_VEL
LIN {X 0,Y 262.869,Z 746.133,A -85,B 0,C 180,E1 -18086.168,E2 -18086.168} C_VEL
LIN {X 0,Y 263.2,Z 749.013,A -85,B 0,C 180,E1 -18088.47,E2 -18088.47} C_VEL
LIN {X 0,Y 263.477,Z 750.163,A -85,B 0,C 180,E1 -18090,E2 -18090} C_VEL
LIN {X 0,Y 262.948,Z 750.65,A -85,B 0,C 180,E1 -18091.531,E2 -18091.531} C_VEL
LIN {X 0,Y 262.536,Z 750.576,A -85,B 0,C 180,E1 -18093.069,E2 -18093.069} C_VEL
LIN {X 0,Y 262.232,Z 750.019,A -85,B 0,C 180,E1 -18094.611,E2 -18094.611} C_VEL
LIN {X 0,Y 261.842,Z 748.38,A -85,B 0,C 180,E1 -18096.737,E2 -18096.737} C_VEL
LIN {X 0,Y 261.892,Z 745.185,A -85,B 0,C 180,E1 -18099.265,E2 -18099.265} C_VEL
LIN {X 0,Y 262.369,Z 740.989,A -85,B 0,C 180,E1 -18101.589,E2 -18101.589} C_VEL
LIN {X 0,Y 263.508,Z 735.491,A -85,B 0,C 180,E1 -18103.888,E2 -18103.888} C_VEL
LIN {X 0,Y 265.327,Z 728.498,A -85,B 0,C 180,E1 -18106.148,E2 -18106.148} C_VEL
LIN {X 0,Y 267.138,Z 721.295,A -85,B 0,C 180,E1 -18108.006,E2 -18108.006} C_VEL
LIN {X 0,Y 269.548,Z 712.45,A -85,B 0,C 180,E1 -18109.812,E2 -18109.812} C_VEL
LIN {X 0,Y 272.084,Z 702.687,A -85,B 0,C 180,E1 -18111.403,E2 -18111.403} C_VEL
LIN {X 0,Y 274.84,Z 690.605,A -85,B 0,C 180,E1 -18112.951,E2 -18112.951} C_VEL
LIN {X 0,Y 277.455,Z 677.391,A -85,B 0,C 180,E1 -18114.206,E2 -18114.206} C_VEL
LIN {X 0,Y 279.511,Z 664.159,A -85,B 0,C 180,E1 -18115.106,E2 -18115.106} C_VEL
LIN {X 0,Y 280.405,Z 653.104,A -85,B 0,C 180,E1 -18115.686,E2 -18115.686} C_VEL
LIN {X 0,Y 280.223,Z 632.214,A -85,B 0,C 180,E1 -18116.707,E2 -18116.707} C_VEL
LIN {X 0,Y 279.23,Z 617.797,A -85,B 0,C 180,E1 -18117.59,E2 -18117.59} C_VEL
LIN {X 0,Y 277.481,Z 602.691,A -85,B 0,C 180,E1 -18118.668,E2 -18118.668} C_VEL
LIN {X 0,Y 275.045,Z 587.678,A -85,B 0,C 180,E1 -18119.946,E2 -18119.946} C_VEL
LIN {X 0,Y 272.367,Z 574.387,A -85,B 0,C 180,E1 -18121.266,E2 -18121.266} C_VEL
LIN {X 0,Y 271.097,Z 569.217,A -85,B 0,C 180,E1 -18121.855,E2 -18121.855} C_VEL
LIN {X 0,Y 269.478,Z 564.733,A -85,B 0,C 180,E1 -18122.52,E2 -18122.52} C_VEL
LIN {X 0,Y 266.912,Z 559.205,A -85,B 0,C 180,E1 -18123.544,E2 -18123.544} C_VEL
LIN {X 0,Y 266.417,Z 557.291,A -85,B 0,C 180,E1 -18123.956,E2 -18123.956} C_VEL
LIN {X 0,Y 264.89,Z 549.919,A -85,B 0,C 180,E1 -18127.255,E2 -18127.255} C_VEL
LIN {X 0,Y 263.165,Z 542.668,A -85,B 0,C 180,E1 -18130.991,E2 -18130.991} C_VEL
LIN {X 0,Y 263.134,Z 542.517,A -85,B 0,C 180,E1 -18133.98,E2 -18133.98} C_VEL
LIN {X 0,Y 263.206,Z 542.504,A -85,B 0,C 180,E1 -18138.385,E2 -18138.385} C_VEL
LIN {X 0,Y 263.202,Z 542.508,A -85,B 0,C 180,E1 -18143.229,E2 -18143.229} C_VEL
LIN {X 0,Y 263.179,Z 542.516,A -85,B 0,C 180,E1 -18145.89,E2 -18145.89} C_VEL
LIN {X 0,Y 263.136,Z 542.519,A -85,B 0,C 180,E1 -18149.505,E2 -18149.505} C_VEL
LIN {X 0,Y 263.186,Z 542.508,A -85,B 0,C 180,E1 -18153.003,E2 -18153.003} C_VEL
LIN {X 0,Y 263.179,Z 542.508,A -85,B 0,C 180,E1 -18156.387,E2 -18156.387} C_VEL
LIN {X 0,Y 263.258,Z 542.498,A -85,B 0,C 180,E1 -18159.693,E2 -18159.693} C_VEL
LIN {X 0,Y 263.338,Z 542.49,A -85,B 0,C 180,E1 -18164.522,E2 -18164.522} C_VEL
LIN {X 0,Y 263.358,Z 542.807,A -85,B 0,C 180,E1 -18165.562,E2 -18165.562} C_VEL
LIN {X 0,Y 263.689,Z 544.092,A -85,B 0,C 180,E1 -18165.949,E2 -18165.949} C_VEL
LIN {X 0,Y 265.37,Z 546.661,A -85,B 0,C 180,E1 -18166.612,E2 -18166.612} C_VEL
LIN {X 0,Y 266.954,Z 548.189,A -85,B 0,C 180,E1 -18167.144,E2 -18167.144} C_VEL
LIN {X 0,Y 269,Z 551.393,A -85,B 0,C 180,E1 -18167.883,E2 -18167.883} C_VEL
LIN {X 0,Y 270.417,Z 553.095,A -85,B 0,C 180,E1 -18168.346,E2 -18168.346} C_VEL
LIN {X 0,Y 272.671,Z 556.366,A -85,B 0,C 180,E1 -18169.06,E2 -18169.06} C_VEL
LIN {X 0,Y 277.898,Z 564.378,A -85,B 0,C 180,E1 -18170.634,E2 -18170.634} C_VEL
LIN {X 0,Y 285.641,Z 578.768,A -85,B 0,C 180,E1 -18172.779,E2 -18172.779} C_VEL
LIN {X 0,Y 285.288,Z 593.039,A -85,B 0,C 180,E1 -18173.41,E2 -18173.41} C_VEL
LIN {X 0,Y 284.573,Z 604.758,A -85,B 0,C 180,E1 -18174.198,E2 -18174.198} C_VEL
LIN {X 0,Y 283.371,Z 616.034,A -85,B 0,C 180,E1 -18175.207,E2 -18175.207} C_VEL
LIN {X 0,Y 281.634,Z 627.31,A -85,B 0,C 180,E1 -18176.515,E2 -18176.515} C_VEL
LIN {X 0,Y 279.699,Z 637.392,A -85,B 0,C 180,E1 -18178.021,E2 -18178.021} C_VEL
LIN {X 0,Y 277.715,Z 646.156,A -85,B 0,C 180,E1 -18179.638,E2 -18179.638} C_VEL
LIN {X 0,Y 275.527,Z 654.098,A -85,B 0,C 180,E1 -18181.462,E2 -18181.462} C_VEL
LIN {X 0,Y 273.148,Z 661.744,A -85,B 0,C 180,E1 -18183.689,E2 -18183.689} C_VEL
LIN {X 0,Y 271,Z 667.693,A -85,B 0,C 180,E1 -18185.955,E2 -18185.955} C_VEL
LIN {X 0,Y 269.162,Z 672.137,A -85,B 0,C 180,E1 -18188.182,E2 -18188.182} C_VEL
LIN {X 0,Y 267.515,Z 675.633,A -85,B 0,C 180,E1 -18190.598,E2 -18190.598} C_VEL
LIN {X 0,Y 266.369,Z 677.509,A -85,B 0,C 180,E1 -18192.526,E2 -18192.526} C_VEL
LIN {X 0,Y 265.092,Z 678.956,A -85,B 0,C 180,E1 -18195.374,E2 -18195.374} C_VEL
LIN {X 0,Y 264.53,Z 679.064,A -85,B 0,C 180,E1 -18196.993,E2 -18196.993} C_VEL
LIN {X 0,Y 264.079,Z 678.729,A -85,B 0,C 180,E1 -18198.625,E2 -18198.625} C_VEL
LIN {X 0,Y 263.659,Z 677.246,A -85,B 0,C 180,E1 -18201.105,E2 -18201.105} C_VEL
LIN {X 0,Y 263.508,Z 674.609,A -85,B 0,C 180,E1 -18203.583,E2 -18203.583} C_VEL
LIN {X 0,Y 263.694,Z 670.707,A -85,B 0,C 180,E1 -18206.089,E2 -18206.089} C_VEL
LIN {X 0,Y 264.023,Z 665.387,A -85,B 0,C 180,E1 -18208.63,E2 -18208.63} C_VEL
LIN {X 0,Y 264.66,Z 658.325,A -85,B 0,C 180,E1 -18211.187,E2 -18211.187} C_VEL
LIN {X 0,Y 265.411,Z 650.906,A -85,B 0,C 180,E1 -18213.33,E2 -18213.33} C_VEL
LIN {X 0,Y 266.326,Z 641.554,A -85,B 0,C 180,E1 -18215.49,E2 -18215.49} C_VEL
LIN {X 0,Y 267.202,Z 632.296,A -85,B 0,C 180,E1 -18217.226,E2 -18217.226} C_VEL
LIN {X 0,Y 268.117,Z 621.768,A -85,B 0,C 180,E1 -18218.822,E2 -18218.822} C_VEL
LIN {X 0,Y 268.938,Z 609.436,A -85,B 0,C 180,E1 -18220.3,E2 -18220.3} C_VEL
LIN {X 0,Y 269.642,Z 597.227,A -85,B 0,C 180,E1 -18221.405,E2 -18221.405} C_VEL
LIN {X 0,Y 270.111,Z 583.814,A -85,B 0,C 180,E1 -18222.284,E2 -18222.284} C_VEL
LIN {X 0,Y 270.245,Z 568.824,A -85,B 0,C 180,E1 -18222.902,E2 -18222.902} C_VEL
LIN {X 0,Y 270.119,Z 564.633,A -85,B 0,C 180,E1 -18223.056,E2 -18223.056} C_VEL
LIN {X 0,Y 263.363,Z 543.528,A -85,B 0,C 180,E1 -18224.168,E2 -18224.168} C_VEL
LIN {X 0,Y 263.208,Z 542.654,A -85,B 0,C 180,E1 -18224.419,E2 -18224.419} C_VEL
LIN {X 0,Y 263.173,Z 542.514,A -85,B 0,C 180,E1 -18228.396,E2 -18228.396} C_VEL
LIN {X 0,Y 263.189,Z 542.512,A -85,B 0,C 180,E1 -18232.109,E2 -18232.109} C_VEL
LIN {X 0,Y 263.185,Z 542.513,A -85,B 0,C 180,E1 -18235.892,E2 -18235.892} C_VEL
LIN {X 0,Y 263.153,Z 542.52,A -85,B 0,C 180,E1 -18239.508,E2 -18239.508} C_VEL
LIN {X 0,Y 263.195,Z 542.511,A -85,B 0,C 180,E1 -18243.004,E2 -18243.004} C_VEL
LIN {X 0,Y 263.185,Z 542.511,A -85,B 0,C 180,E1 -18246.388,E2 -18246.388} C_VEL
LIN {X 0,Y 263.255,Z 542.506,A -85,B 0,C 180,E1 -18249.693,E2 -18249.693} C_VEL
LIN {X 0,Y 263.318,Z 542.493,A -85,B 0,C 180,E1 -18254.521,E2 -18254.521} C_VEL
LIN {X 0,Y 263.358,Z 542.491,A -85,B 0,C 180,E1 -18259.234,E2 -18259.234} C_VEL
LIN {X 0,Y 263.537,Z 542.466,A -85,B 0,C 180,E1 -18262.338,E2 -18262.338} C_VEL
LIN {X 0,Y 263.755,Z 542.44,A -85,B 0,C 180,E1 -18268.473,E2 -18268.473} C_VEL
LIN {X 0,Y 263.755,Z 542.442,A -85,B 0,C 180,E1 -18271.527,E2 -18271.527} C_VEL
LIN {X 0,Y 263.537,Z 542.471,A -85,B 0,C 180,E1 -18277.663,E2 -18277.663} C_VEL
LIN {X 0,Y 263.357,Z 542.488,A -85,B 0,C 180,E1 -18280.766,E2 -18280.766} C_VEL
LIN {X 0,Y 263.355,Z 542.492,A -85,B 0,C 180,E1 -18285.477,E2 -18285.477} C_VEL
LIN {X 0,Y 263.266,Z 542.502,A -85,B 0,C 180,E1 -18290.306,E2 -18290.306} C_VEL
LIN {X 0,Y 263.195,Z 542.51,A -85,B 0,C 180,E1 -18295.292,E2 -18295.292} C_VEL
LIN {X 0,Y 263.168,Z 542.512,A -85,B 0,C 180,E1 -18298.73,E2 -18298.73} C_VEL
LIN {X 0,Y 263.135,Z 542.52,A -85,B 0,C 180,E1 -18302.287,E2 -18302.287} C_VEL
LIN {X 0,Y 263.192,Z 542.514,A -85,B 0,C 180,E1 -18305.976,E2 -18305.976} C_VEL
LIN {X 0,Y 263.161,Z 542.517,A -85,B 0,C 180,E1 -18309.861,E2 -18309.861} C_VEL
LIN {X 0,Y 263.145,Z 542.52,A -85,B 0,C 180,E1 -18313.978,E2 -18313.978} C_VEL
LIN {X 0,Y 263.129,Z 542.521,A -85,B 0,C 180,E1 -18318.404,E2 -18318.404} C_VEL
LIN {X 0,Y 263.192,Z 542.509,A -85,B 0,C 180,E1 -18323.232,E2 -18323.232} C_VEL
LIN {X 0,Y 263.166,Z 542.514,A -85,B 0,C 180,E1 -18325.887,E2 -18325.887} C_VEL
LIN {X 0,Y 263.146,Z 542.517,A -85,B 0,C 180,E1 -18329.506,E2 -18329.506} C_VEL
LIN {X 0,Y 263.189,Z 542.509,A -85,B 0,C 180,E1 -18333.002,E2 -18333.002} C_VEL
LIN {X 0,Y 263.184,Z 542.516,A -85,B 0,C 180,E1 -18336.386,E2 -18336.386} C_VEL
LIN {X 0,Y 263.265,Z 542.502,A -85,B 0,C 180,E1 -18339.693,E2 -18339.693} C_VEL
LIN {X 0,Y 263.341,Z 542.495,A -85,B 0,C 180,E1 -18344.521,E2 -18344.521} C_VEL
LIN {X 0,Y 263.37,Z 542.488,A -85,B 0,C 180,E1 -18349.234,E2 -18349.234} C_VEL
LIN {X 0,Y 263.568,Z 542.466,A -85,B 0,C 180,E1 -18352.338,E2 -18352.338} C_VEL
LIN {X 0,Y 263.746,Z 542.445,A -85,B 0,C 180,E1 -18358.473,E2 -18358.473} C_VEL
LIN {X 0,Y 263.746,Z 542.44,A -85,B 0,C 180,E1 -18361.526,E2 -18361.526} C_VEL
LIN {X 0,Y 263.564,Z 542.463,A -85,B 0,C 180,E1 -18367.661,E2 -18367.661} C_VEL
LIN {X 0,Y 263.368,Z 542.491,A -85,B 0,C 180,E1 -18370.765,E2 -18370.765} C_VEL
LIN {X 0,Y 263.339,Z 542.492,A -85,B 0,C 180,E1 -18375.478,E2 -18375.478} C_VEL
LIN {X 0,Y 263.257,Z 542.503,A -85,B 0,C 180,E1 -18380.307,E2 -18380.307} C_VEL
LIN {X 0,Y 263.199,Z 542.512,A -85,B 0,C 180,E1 -18380.941,E2 -18380.941} C_VEL
LIN {X 0,Y 262.439,Z 542.608,A -85,B 0,C 180,E1 -18382.219,E2 -18382.219} C_VEL
LIN {X 0,Y 259.53,Z 542.969,A -85,B 0,C 180,E1 -18384.302,E2 -18384.302} C_VEL
LIN {X 0,Y 257.149,Z 543.262,A -85,B 0,C 180,E1 -18385.996,E2 -18385.996} C_VEL
LIN {X 0,Y 256.185,Z 543.382,A -85,B 0,C 180,E1 -18387.31,E2 -18387.31} C_VEL
LIN {X 0,Y 256.134,Z 543.388,A -85,B 0,C 180,E1 -18387.754,E2 -18387.754} C_VEL
LIN {X 0,Y 256.078,Z 543.397,A -85,B 0,C 180,E1 -18391.704,E2 -18391.704} C_VEL
LIN {X 0,Y 256.077,Z 543.396,A -85,B 0,C 180,E1 -18395.193,E2 -18395.193} C_VEL
LIN {X 0,Y 256.109,Z 543.393,A -85,B 0,C 180,E1 -18397.271,E2 -18397.271} C_VEL
LIN {X 0,Y 256.051,Z 543.402,A -85,B 0,C 180,E1 -18401.204,E2 -18401.204} C_VEL
LIN {X 0,Y 256.058,Z 543.4,A -85,B 0,C 180,E1 -18405.529,E2 -18405.529} C_VEL
LIN {X 0,Y 256.054,Z 543.404,A -85,B 0,C 180,E1 -18408.798,E2 -18408.798} C_VEL
LIN {X 0,Y 256.269,Z 543.503,A -85,B 0,C 180,E1 -18413.383,E2 -18413.383} C_VEL
LIN {X 0,Y 258.696,Z 556.081,A -85,B 0,C 180,E1 -18418.248,E2 -18418.248} C_VEL
LIN {X 0,Y 259.447,Z 559.822,A -85,B 0,C 180,E1 -18419.636,E2 -18419.636} C_VEL
LIN {X 0,Y 258.392,Z 567.728,A -85,B 0,C 180,E1 -18422.46,E2 -18422.46} C_VEL
LIN {X 0,Y 256.627,Z 581.354,A -85,B 0,C 180,E1 -18427.243,E2 -18427.243} C_VEL
LIN {X 0,Y 257.203,Z 596.038,A -85,B 0,C 180,E1 -18427.949,E2 -18427.949} C_VEL
LIN {X 0,Y 260.852,Z 654.35,A -85,B 0,C 180,E1 -18430.547,E2 -18430.547} C_VEL
LIN {X 0,Y 260.278,Z 670.594,A -85,B 0,C 180,E1 -18431.298,E2 -18431.298} C_VEL
LIN {X 0,Y 259.52,Z 683.71,A -85,B 0,C 180,E1 -18432.263,E2 -18432.263} C_VEL
LIN {X 0,Y 258.486,Z 694.889,A -85,B 0,C 180,E1 -18433.412,E2 -18433.412} C_VEL
LIN {X 0,Y 257.439,Z 705.022,A -85,B 0,C 180,E1 -18434.766,E2 -18434.766} C_VEL
LIN {X 0,Y 256.65,Z 714.327,A -85,B 0,C 180,E1 -18436.339,E2 -18436.339} C_VEL
LIN {X 0,Y 255.922,Z 722.735,A -85,B 0,C 180,E1 -18438.114,E2 -18438.114} C_VEL
LIN {X 0,Y 255.475,Z 730.259,A -85,B 0,C 180,E1 -18440.1,E2 -18440.1} C_VEL
LIN {X 0,Y 255.388,Z 736.497,A -85,B 0,C 180,E1 -18442.169,E2 -18442.169} C_VEL
LIN {X 0,Y 255.618,Z 741.857,A -85,B 0,C 180,E1 -18444.478,E2 -18444.478} C_VEL
LIN {X 0,Y 255.931,Z 745.841,A -85,B 0,C 180,E1 -18446.852,E2 -18446.852} C_VEL
LIN {X 0,Y 256.203,Z 747.685,A -85,B 0,C 180,E1 -18448.428,E2 -18448.428} C_VEL
LIN {X 0,Y 256.476,Z 748.94,A -85,B 0,C 180,E1 -18450,E2 -18450} C_VEL
LIN {X 0,Y 255.93,Z 749.478,A -85,B 0,C 180,E1 -18451.573,E2 -18451.573} C_VEL
LIN {X 0,Y 255.477,Z 749.496,A -85,B 0,C 180,E1 -18453.154,E2 -18453.154} C_VEL
LIN {X 0,Y 255.163,Z 748.997,A -85,B 0,C 180,E1 -18454.74,E2 -18454.74} C_VEL
LIN {X 0,Y 254.775,Z 747.621,A -85,B 0,C 180,E1 -18456.756,E2 -18456.756} C_VEL
LIN {X 0,Y 254.834,Z 744.449,A -85,B 0,C 180,E1 -18459.524,E2 -18459.524} C_VEL
LIN {X 0,Y 255.36,Z 740.415,A -85,B 0,C 180,E1 -18461.912,E2 -18461.912} C_VEL
LIN {X 0,Y 256.593,Z 735.128,A -85,B 0,C 180,E1 -18464.27,E2 -18464.27} C_VEL
LIN {X 0,Y 258.495,Z 728.356,A -85,B 0,C 180,E1 -18466.587,E2 -18466.587} C_VEL
LIN {X 0,Y 260.871,Z 719.821,A -85,B 0,C 180,E1 -18468.861,E2 -18468.861} C_VEL
LIN {X 0,Y 263.488,Z 711.007,A -85,B 0,C 180,E1 -18470.696,E2 -18470.696} C_VEL
LIN {X 0,Y 266.171,Z 701.108,A -85,B 0,C 180,E1 -18472.343,E2 -18472.343} C_VEL
LIN {X 0,Y 268.714,Z 690.655,A -85,B 0,C 180,E1 -18473.71,E2 -18473.71} C_VEL
LIN {X 0,Y 271.239,Z 678.862,A -85,B 0,C 180,E1 -18474.9,E2 -18474.9} C_VEL
LIN {X 0,Y 273.59,Z 665.472,A -85,B 0,C 180,E1 -18475.893,E2 -18475.893} C_VEL
LIN {X 0,Y 274.737,Z 654.606,A -85,B 0,C 180,E1 -18476.52,E2 -18476.52} C_VEL
LIN {X 0,Y 274.81,Z 633.758,A -85,B 0,C 180,E1 -18477.598,E2 -18477.598} C_VEL
LIN {X 0,Y 273.9,Z 619.404,A -85,B 0,C 180,E1 -18478.5,E2 -18478.5} C_VEL
LIN {X 0,Y 272.263,Z 604.054,A -85,B 0,C 180,E1 -18479.646,E2 -18479.646} C_VEL
LIN {X 0,Y 269.492,Z 586.531,A -85,B 0,C 180,E1 -18481.235,E2 -18481.235} C_VEL
LIN {X 0,Y 266.894,Z 573.543,A -85,B 0,C 180,E1 -18482.644,E2 -18482.644} C_VEL
LIN {X 0,Y 265.283,Z 569.136,A -85,B 0,C 180,E1 -18483.337,E2 -18483.337} C_VEL
LIN {X 0,Y 262.634,Z 562.922,A -85,B 0,C 180,E1 -18484.477,E2 -18484.477} C_VEL
LIN {X 0,Y 259.22,Z 556.031,A -85,B 0,C 180,E1 -18486.017,E2 -18486.017} C_VEL
LIN {X 0,Y 258.529,Z 553.867,A -85,B 0,C 180,E1 -18486.523,E2 -18486.523} C_VEL
LIN {X 0,Y 257.283,Z 548.353,A -85,B 0,C 180,E1 -18489.186,E2 -18489.186} C_VEL
LIN {X 0,Y 256.107,Z 543.464,A -85,B 0,C 180,E1 -18491.938,E2 -18491.938} C_VEL
LIN {X 0,Y 256.107,Z 543.394,A -85,B 0,C 180,E1 -18496.683,E2 -18496.683} C_VEL
LIN {X 0,Y 256.104,Z 543.388,A -85,B 0,C 180,E1 -18500.864,E2 -18500.864} C_VEL
LIN {X 0,Y 256.117,Z 543.387,A -85,B 0,C 180,E1 -18504.813,E2 -18504.813} C_VEL
LIN {X 0,Y 256.087,Z 543.395,A -85,B 0,C 180,E1 -18508.572,E2 -18508.572} C_VEL
LIN {X 0,Y 256.133,Z 543.394,A -85,B 0,C 180,E1 -18512.196,E2 -18512.196} C_VEL
LIN {X 0,Y 256.162,Z 543.387,A -85,B 0,C 180,E1 -18515.699,E2 -18515.699} C_VEL
LIN {X 0,Y 256.163,Z 543.383,A -85,B 0,C 180,E1 -18519.105,E2 -18519.105} C_VEL
LIN {X 0,Y 256.25,Z 543.56,A -85,B 0,C 180,E1 -18523.089,E2 -18523.089} C_VEL
LIN {X 0,Y 256.473,Z 544.442,A -85,B 0,C 180,E1 -18523.549,E2 -18523.549} C_VEL
LIN {X 0,Y 258.199,Z 547.382,A -85,B 0,C 180,E1 -18524.408,E2 -18524.408} C_VEL
LIN {X 0,Y 260.242,Z 549.276,A -85,B 0,C 180,E1 -18525.214,E2 -18525.214} C_VEL
LIN {X 0,Y 262.16,Z 552.47,A -85,B 0,C 180,E1 -18526.039,E2 -18526.039} C_VEL
LIN {X 0,Y 263.851,Z 554.364,A -85,B 0,C 180,E1 -18526.644,E2 -18526.644} C_VEL
LIN {X 0,Y 266.308,Z 557.817,A -85,B 0,C 180,E1 -18527.533,E2 -18527.533} C_VEL
LIN {X 0,Y 271.11,Z 564.928,A -85,B 0,C 180,E1 -18529.133,E2 -18529.133} C_VEL
LIN {X 0,Y 275.077,Z 571.679,A -85,B 0,C 180,E1 -18530.39,E2 -18530.39} C_VEL
LIN {X 0,Y 280.37,Z 581.879,A -85,B 0,C 180,E1 -18531.932,E2 -18531.932} C_VEL
LIN {X 0,Y 279.89,Z 595.44,A -85,B 0,C 180,E1 -18532.572,E2 -18532.572} C_VEL
LIN {X 0,Y 278.948,Z 607.694,A -85,B 0,C 180,E1 -18533.448,E2 -18533.448} C_VEL
LIN {X 0,Y 277.568,Z 619.175,A -85,B 0,C 180,E1 -18534.532,E2 -18534.532} C_VEL
LIN {X 0,Y 275.819,Z 629.671,A -85,B 0,C 180,E1 -18535.818,E2 -18535.818} C_VEL
LIN {X 0,Y 273.643,Z 640.041,A -85,B 0,C 180,E1 -18537.424,E2 -18537.424} C_VEL
LIN {X 0,Y 271.293,Z 649.282,A -85,B 0,C 180,E1 -18539.258,E2 -18539.258} C_VEL
LIN {X 0,Y 268.971,Z 656.869,A -85,B 0,C 180,E1 -18541.123,E2 -18541.123} C_VEL
LIN {X 0,Y 266.907,Z 663.072,A -85,B 0,C 180,E1 -18543.019,E2 -18543.019} C_VEL
LIN {X 0,Y 264.59,Z 669.01,A -85,B 0,C 180,E1 -18545.335,E2 -18545.335} C_VEL
LIN {X 0,Y 262.465,Z 673.757,A -85,B 0,C 180,E1 -18547.812,E2 -18547.812} C_VEL
LIN {X 0,Y 261.406,Z 675.898,A -85,B 0,C 180,E1 -18549.284,E2 -18549.284} C_VEL
LIN {X 0,Y 260.339,Z 677.691,A -85,B 0,C 180,E1 -18550.893,E2 -18550.893} C_VEL
LIN {X 0,Y 259.307,Z 679.124,A -85,B 0,C 180,E1 -18552.662,E2 -18552.662} C_VEL
LIN {X 0,Y 258.565,Z 679.852,A -85,B 0,C 180,E1 -18554.16,E2 -18554.16} C_VEL
LIN {X 0,Y 257.901,Z 680.213,A -85,B 0,C 180,E1 -18555.814,E2 -18555.814} C_VEL
LIN {X 0,Y 257.375,Z 680.068,A -85,B 0,C 180,E1 -18557.481,E2 -18557.481} C_VEL
LIN {X 0,Y 256.944,Z 679.435,A -85,B 0,C 180,E1 -18559.162,E2 -18559.162} C_VEL
LIN {X 0,Y 256.579,Z 677.86,A -85,B 0,C 180,E1 -18561.365,E2 -18561.365} C_VEL
LIN {X 0,Y 256.468,Z 674.477,A -85,B 0,C 180,E1 -18564.271,E2 -18564.271} C_VEL
LIN {X 0,Y 256.701,Z 670.07,A -85,B 0,C 180,E1 -18566.856,E2 -18566.856} C_VEL
LIN {X 0,Y 257.142,Z 664.19,A -85,B 0,C 180,E1 -18569.47,E2 -18569.47} C_VEL
LIN {X 0,Y 257.767,Z 657.406,A -85,B 0,C 180,E1 -18571.81,E2 -18571.81} C_VEL
LIN {X 0,Y 258.52,Z 650.019,A -85,B 0,C 180,E1 -18573.87,E2 -18573.87} C_VEL
LIN {X 0,Y 259.473,Z 640.673,A -85,B 0,C 180,E1 -18575.994,E2 -18575.994} C_VEL
LIN {X 0,Y 260.436,Z 630.303,A -85,B 0,C 180,E1 -18577.874,E2 -18577.874} C_VEL
LIN {X 0,Y 261.338,Z 619.533,A -85,B 0,C 180,E1 -18579.448,E2 -18579.448} C_VEL
LIN {X 0,Y 262.128,Z 607.767,A -85,B 0,C 180,E1 -18580.795,E2 -18580.795} C_VEL
LIN {X 0,Y 262.813,Z 595.445,A -85,B 0,C 180,E1 -18581.87,E2 -18581.87} C_VEL
LIN {X 0,Y 263.186,Z 582.313,A -85,B 0,C 180,E1 -18582.68,E2 -18582.68} C_VEL
LIN {X 0,Y 263.163,Z 565.829,A -85,B 0,C 180,E1 -18583.34,E2 -18583.34} C_VEL
LIN {X 0,Y 256.3,Z 544.29,A -85,B 0,C 180,E1 -18584.527,E2 -18584.527} C_VEL
LIN {X 0,Y 256.147,Z 543.446,A -85,B 0,C 180,E1 -18584.86,E2 -18584.86} C_VEL
LIN {X 0,Y 256.103,Z 543.396,A -85,B 0,C 180,E1 -18588.807,E2 -18588.807} C_VEL
LIN {X 0,Y 256.156,Z 543.389,A -85,B 0,C 180,E1 -18592.873,E2 -18592.873} C_VEL
LIN {X 0,Y 256.086,Z 543.396,A -85,B 0,C 180,E1 -18596.711,E2 -18596.711} C_VEL
LIN {X 0,Y 256.14,Z 543.393,A -85,B 0,C 180,E1 -18601.406,E2 -18601.406} C_VEL
LIN {X 0,Y 256.169,Z 543.388,A -85,B 0,C 180,E1 -18605.7,E2 -18605.7} C_VEL
LIN {X 0,Y 256.165,Z 543.387,A -85,B 0,C 180,E1 -18609.105,E2 -18609.105} C_VEL
LIN {X 0,Y 256.251,Z 543.375,A -85,B 0,C 180,E1 -18614.082,E2 -18614.082} C_VEL
LIN {X 0,Y 256.294,Z 543.372,A -85,B 0,C 180,E1 -18617.328,E2 -18617.328} C_VEL
LIN {X 0,Y 256.499,Z 543.343,A -85,B 0,C 180,E1 -18622.126,E2 -18622.126} C_VEL
LIN {X 0,Y 256.499,Z 543.344,A -85,B 0,C 180,E1 -18626.859,E2 -18626.859} C_VEL
LIN {X 0,Y 256.77,Z 543.311,A -85,B 0,C 180,E1 -18630,E2 -18630} C_VEL
LIN {X 0,Y 256.5,Z 543.344,A -85,B 0,C 180,E1 -18633.141,E2 -18633.141} C_VEL
LIN {X 0,Y 256.499,Z 543.347,A -85,B 0,C 180,E1 -18637.874,E2 -18637.874} C_VEL
LIN {X 0,Y 256.298,Z 543.369,A -85,B 0,C 180,E1 -18642.672,E2 -18642.672} C_VEL
LIN {X 0,Y 256.287,Z 543.372,A -85,B 0,C 180,E1 -18646.302,E2 -18646.302} C_VEL
LIN {X 0,Y 256.157,Z 543.386,A -85,B 0,C 180,E1 -18651.117,E2 -18651.117} C_VEL
LIN {X 0,Y 256.173,Z 543.385,A -85,B 0,C 180,E1 -18655.129,E2 -18655.129} C_VEL
LIN {X 0,Y 256.106,Z 543.393,A -85,B 0,C 180,E1 -18659.6,E2 -18659.6} C_VEL
LIN {X 0,Y 256.087,Z 543.396,A -85,B 0,C 180,E1 -18663.289,E2 -18663.289} C_VEL
LIN {X 0,Y 256.142,Z 543.386,A -85,B 0,C 180,E1 -18667.278,E2 -18667.278} C_VEL
LIN {X 0,Y 256.105,Z 543.393,A -85,B 0,C 180,E1 -18671.193,E2 -18671.193} C_VEL
LIN {X 0,Y 256.072,Z 543.396,A -85,B 0,C 180,E1 -18675.526,E2 -18675.526} C_VEL
LIN {X 0,Y 256.058,Z 543.4,A -85,B 0,C 180,E1 -18678.796,E2 -18678.796} C_VEL
LIN {X 0,Y 256.137,Z 543.389,A -85,B 0,C 180,E1 -18682.868,E2 -18682.868} C_VEL
LIN {X 0,Y 256.075,Z 543.398,A -85,B 0,C 180,E1 -18686.707,E2 -18686.707} C_VEL
LIN {X 0,Y 256.133,Z 543.389,A -85,B 0,C 180,E1 -18691.405,E2 -18691.405} C_VEL
LIN {X 0,Y 256.165,Z 543.386,A -85,B 0,C 180,E1 -18695.698,E2 -18695.698} C_VEL
LIN {X 0,Y 256.215,Z 543.38,A -85,B 0,C 180,E1 -18699.108,E2 -18699.108} C_VEL
LIN {X 0,Y 256.291,Z 543.371,A -85,B 0,C 180,E1 -18704.084,E2 -18704.084} C_VEL
